Universal Robots PolyScope program: jerry_robot_1.urp

Program jerry_robot_1 (installation=default directory=/programs createdIn=5.11.9.1010452 lastSavedIn=5.11.9.1010452 robotSerialNumber=20225200364)
Calibrated DH parameters: a=[0.00002, -0.569483, -0.54992, -0.00001, -0.000036, 0]; d=[0.180894, -146.691669, 192.918669, -46.053088, 0.119778, 0.115602]; alpha=[1.571425, -0.001534, 0.003359, 1.568739, -1.571477, 0]; deltaTheta=[0, 0.376258, -0.101074, -0.275185, -0.000002, 0]
Robot Program (runOnlyOnce=false)
  Script file /programs/usbdisk/UR/jerry_new_robot_2.script
    | def Machining2():
    |   # Default parameters:
    |   global speed_ms = 0.3
    |   global speed_rads = 0.75
    |   global accel_mss = 3
    |   global accel_radss = 1.2
    |   global blend_radius_m = 0.0003
    | 
    |   # Add subprograms here
    |   # Start of main program
    |   # Program generated by RoboDK v5.6.8 for UR10e on 15/12/2023 16:19:10
    |   # Using nominal kinematics.
    |   blend_radius_m = 0.0003
    |   speed_ms = 0.01
    |   # set_reference(p[0.405000, -0.105000, 0.002000, 0.000000, 0.000000, 0.000000])
    |   set_tcp(p[0.000000, 0.000000, 0.252000, 0.000000, 0.000000, 0.000000])
    |   # Show Tool
    |   movej([0.340820, -1.401012, -2.442590, -0.868787, 1.570796, 1.911616],accel_radss,speed_rads,0,blend_radius_m)
    |   movel([0.340820, -1.453448, -2.472410, -0.786531, 1.570796, 1.911616],accel_mss,speed_ms,0,blend_radius_m)
    |   speed_ms = 0.01
    |   movel([0.340820, -1.476287, -2.483478, -0.752624, 1.570796, 1.911616],accel_mss,speed_ms,0,blend_radius_m)
    |   speed_ms = 0.003
    |   movel([0.340820, -1.485129, -2.487495, -0.739765, 1.570796, 1.911616],accel_mss,speed_ms,0,blend_radius_m)
    |   speed_ms = 0.007
    |   movel([0.329121, -1.487754, -2.485222, -0.739413, 1.570796, 1.899918],accel_mss,speed_ms,0,blend_radius_m)
    |   movel([0.326624, -1.484406, -2.488119, -0.739864, 1.570796, 1.897421],accel_mss,speed_ms,0,blend_radius_m)
    |   movel([0.324102, -1.481056, -2.491001, -0.740332, 1.570796, 1.894899],accel_mss,speed_ms,0,blend_radius_m)
    |   movel([0.325153, -1.479428, -2.492395, -0.740566, 1.570796, 1.895949],accel_mss,speed_ms,0,blend_radius_m)
    |   movel([0.326209, -1.477797, -2.493787, -0.740805, 1.570796, 1.897005],accel_mss,speed_ms,0,blend_radius_m)
    |   movel([0.325032, -1.477528, -2.494017, -0.740845, 1.570796, 1.895828],accel_mss,speed_ms,0,blend_radius_m)
    |   movel([0.324303, -1.477370, -2.494151, -0.740868, 1.570796, 1.895099],accel_mss,speed_ms,0,blend_radius_m)
    |   movel([0.315110, -1.475621, -2.495639, -0.741130, 1.570796, 1.885906],accel_mss,speed_ms,0,blend_radius_m)
    |   movel([0.311619, -1.474970, -2.496191, -0.741228, 1.570796, 1.882415],accel_mss,speed_ms,0,blend_radius_m)
    |   movel([0.310032, -1.474668, -2.496447, -0.741274, 1.570796, 1.880828],accel_mss,speed_ms,0,blend_radius_m)
    |   movel([0.308452, -1.474355, -2.496712, -0.741322, 1.570796, 1.879249],accel_mss,speed_ms,0,blend_radius_m)
    |   movel([0.306876, -1.474033, -2.496985, -0.741371, 1.570796, 1.877673],accel_mss,speed_ms,0,blend_radius_m)
    |   movel([0.305660, -1.473769, -2.497208, -0.741412, 1.570796, 1.876456],accel_mss,speed_ms,0,blend_radius_m)
    |   movel([0.304453, -1.473494, -2.497441, -0.741454, 1.570796, 1.875249],accel_mss,speed_ms,0,blend_radius_m)
    |   movel([0.303253, -1.473205, -2.497685, -0.741499, 1.570796, 1.874050],accel_mss,speed_ms,0,blend_radius_m)
    |   movel([0.302430, -1.472998, -2.497860, -0.741531, 1.570796, 1.873226],accel_mss,speed_ms,0,blend_radius_m)
    |   movel([0.301614, -1.472780, -2.498045, -0.741565, 1.570796, 1.872410],accel_mss,speed_ms,0,blend_radius_m)
    |   movel([0.300804, -1.472554, -2.498235, -0.741600, 1.570796, 1.871600],accel_mss,speed_ms,0,blend_radius_m)
    |   movel([0.299999, -1.472319, -2.498434, -0.741636, 1.570796, 1.870795],accel_mss,speed_ms,0,blend_radius_m)
    |   movel([0.299265, -1.472091, -2.498626, -0.741672, 1.570796, 1.870061],accel_mss,speed_ms,0,blend_radius_m)
    |   movel([0.298537, -1.471853, -2.498826, -0.741709, 1.570796, 1.869333],accel_mss,speed_ms,0,blend_radius_m)
    |   movel([0.297819, -1.471604, -2.499036, -0.741748, 1.570796, 1.868615],accel_mss,speed_ms,0,blend_radius_m)
    |   movel([0.297109, -1.471344, -2.499256, -0.741789, 1.570796, 1.867905],accel_mss,speed_ms,0,blend_radius_m)
    |   movel([0.296406, -1.471071, -2.499485, -0.741832, 1.570796, 1.867203],accel_mss,speed_ms,0,blend_radius_m)
    |   movel([0.295713, -1.470789, -2.499723, -0.741877, 1.570796, 1.866509],accel_mss,speed_ms,0,blend_radius_m)
    |   movel([0.295027, -1.470496, -2.499970, -0.741924, 1.570796, 1.865823],accel_mss,speed_ms,0,blend_radius_m)
    |   movel([0.294528, -1.470268, -2.500162, -0.741960, 1.570796, 1.865325],accel_mss,speed_ms,0,blend_radius_m)
    |   movel([0.294040, -1.470028, -2.500363, -0.741998, 1.570796, 1.864837],accel_mss,speed_ms,0,blend_radius_m)
    |   movel([0.293562, -1.469778, -2.500573, -0.742038, 1.570796, 1.864358],accel_mss,speed_ms,0,blend_radius_m)
    |   movel([0.293093, -1.469515, -2.500794, -0.742080, 1.570796, 1.863889],accel_mss,speed_ms,0,blend_radius_m)
    |   movel([0.292636, -1.469241, -2.501024, -0.742124, 1.570796, 1.863432],accel_mss,speed_ms,0,blend_radius_m)
    |   movel([0.292189, -1.468954, -2.501264, -0.742170, 1.570796, 1.862986],accel_mss,speed_ms,0,blend_radius_m)
    |   movel([0.291754, -1.468657, -2.501513, -0.742218, 1.570796, 1.862551],accel_mss,speed_ms,0,blend_radius_m)
    |   movel([0.291328, -1.468350, -2.501771, -0.742268, 1.570796, 1.862125],accel_mss,speed_ms,0,blend_radius_m)
    |   movel([0.290973, -1.468072, -2.502004, -0.742313, 1.570796, 1.861769],accel_mss,speed_ms,0,blend_radius_m)
    |   movel([0.290628, -1.467784, -2.502245, -0.742360, 1.570796, 1.861425],accel_mss,speed_ms,0,blend_radius_m)
    |   movel([0.290296, -1.467485, -2.502495, -0.742409, 1.570796, 1.861092],accel_mss,speed_ms,0,blend_radius_m)
    |   movel([0.289978, -1.467174, -2.502755, -0.742460, 1.570796, 1.860774],accel_mss,speed_ms,0,blend_radius_m)
    |   movel([0.289671, -1.466852, -2.503024, -0.742513, 1.570796, 1.860467],accel_mss,speed_ms,0,blend_radius_m)
    |   movel([0.289378, -1.466522, -2.503300, -0.742567, 1.570796, 1.860174],accel_mss,speed_ms,0,blend_radius_m)
    |   movel([0.289096, -1.466178, -2.503587, -0.742624, 1.570796, 1.859893],accel_mss,speed_ms,0,blend_radius_m)
    |   movel([0.288831, -1.465826, -2.503881, -0.742682, 1.570796, 1.859627],accel_mss,speed_ms,0,blend_radius_m)
    |   movel([0.288626, -1.465531, -2.504127, -0.742731, 1.570796, 1.859423],accel_mss,speed_ms,0,blend_radius_m)
    |   movel([0.288435, -1.465229, -2.504378, -0.742782, 1.570796, 1.859231],accel_mss,speed_ms,0,blend_radius_m)
    |   movel([0.288257, -1.464916, -2.504639, -0.742834, 1.570796, 1.859053],accel_mss,speed_ms,0,blend_radius_m)
    |   movel([0.288092, -1.464594, -2.504907, -0.742888, 1.570796, 1.858889],accel_mss,speed_ms,0,blend_radius_m)
    |   movel([0.287941, -1.464265, -2.505180, -0.742944, 1.570796, 1.858737],accel_mss,speed_ms,0,blend_radius_m)
    |   movel([0.287804, -1.463927, -2.505461, -0.743001, 1.570796, 1.858601],accel_mss,speed_ms,0,blend_radius_m)
    |   movel([0.287681, -1.463581, -2.505749, -0.743059, 1.570796, 1.858478],accel_mss,speed_ms,0,blend_radius_m)
    |   movel([0.287573, -1.463229, -2.506041, -0.743119, 1.570796, 1.858369],accel_mss,speed_ms,0,blend_radius_m)
    |   movel([0.287477, -1.462868, -2.506341, -0.743181, 1.570796, 1.858274],accel_mss,speed_ms,0,blend_radius_m)
    |   movel([0.287403, -1.462513, -2.506635, -0.743241, 1.570796, 1.858200],accel_mss,speed_ms,0,blend_radius_m)
    |   movel([0.287345, -1.462148, -2.506937, -0.743304, 1.570796, 1.858141],accel_mss,speed_ms,0,blend_radius_m)
    |   movel([0.287305, -1.461779, -2.507243, -0.743367, 1.570796, 1.858101],accel_mss,speed_ms,0,blend_radius_m)
    |   movel([0.287282, -1.461401, -2.507555, -0.743433, 1.570796, 1.858079],accel_mss,speed_ms,0,blend_radius_m)
    |   movel([0.287278, -1.461018, -2.507872, -0.743499, 1.570796, 1.858075],accel_mss,speed_ms,0,blend_radius_m)
    |   movel([0.287291, -1.460591, -2.508225, -0.743573, 1.570796, 1.858087],accel_mss,speed_ms,0,blend_radius_m)
    |   movel([0.287320, -1.460158, -2.508582, -0.743649, 1.570796, 1.858116],accel_mss,speed_ms,0,blend_radius_m)
    |   movel([0.287362, -1.459724, -2.508940, -0.743725, 1.570796, 1.858158],accel_mss,speed_ms,0,blend_radius_m)
    |   movel([0.287419, -1.459283, -2.509304, -0.743802, 1.570796, 1.858216],accel_mss,speed_ms,0,blend_radius_m)
    |   movel([0.287492, -1.458840, -2.509669, -0.743881, 1.570796, 1.858288],accel_mss,speed_ms,0,blend_radius_m)
    |   movel([0.287580, -1.458381, -2.510046, -0.743962, 1.570796, 1.858377],accel_mss,speed_ms,0,blend_radius_m)
    |   movel([0.287685, -1.457918, -2.510427, -0.744044, 1.570796, 1.858482],accel_mss,speed_ms,0,blend_radius_m)
    |   movel([0.287806, -1.457452, -2.510809, -0.744128, 1.570796, 1.858602],accel_mss,speed_ms,0,blend_radius_m)
    |   movel([0.287939, -1.456985, -2.511192, -0.744211, 1.570796, 1.858736],accel_mss,speed_ms,0,blend_radius_m)
    |   movel([0.288089, -1.456515, -2.511578, -0.744296, 1.570796, 1.858886],accel_mss,speed_ms,0,blend_radius_m)
    |   movel([0.288247, -1.456059, -2.511951, -0.744379, 1.570796, 1.859044],accel_mss,speed_ms,0,blend_radius_m)
    |   movel([0.288421, -1.455602, -2.512326, -0.744462, 1.570796, 1.859217],accel_mss,speed_ms,0,blend_radius_m)
    |   movel([0.288612, -1.455142, -2.512701, -0.744545, 1.570796, 1.859408],accel_mss,speed_ms,0,blend_radius_m)
    |   movel([0.288815, -1.454686, -2.513074, -0.744629, 1.570796, 1.859612],accel_mss,speed_ms,0,blend_radius_m)
    |   movel([0.289034, -1.454228, -2.513449, -0.744713, 1.570796, 1.859831],accel_mss,speed_ms,0,blend_radius_m)
    |   movel([0.289272, -1.453758, -2.513832, -0.744800, 1.570796, 1.860068],accel_mss,speed_ms,0,blend_radius_m)
    |   movel([0.289521, -1.453288, -2.514214, -0.744886, 1.570796, 1.860317],accel_mss,speed_ms,0,blend_radius_m)
    |   movel([0.289777, -1.452822, -2.514594, -0.744973, 1.570796, 1.860573],accel_mss,speed_ms,0,blend_radius_m)
    |   movel([0.290044, -1.452355, -2.514974, -0.745060, 1.570796, 1.860841],accel_mss,speed_ms,0,blend_radius_m)
    |   movel([0.290115, -1.452249, -2.515060, -0.745080, 1.570796, 1.860912],accel_mss,speed_ms,0,blend_radius_m)
    |   movel([0.290197, -1.452143, -2.515146, -0.745100, 1.570796, 1.860993],accel_mss,speed_ms,0,blend_radius_m)
    |   movel([0.290291, -1.452045, -2.515226, -0.745118, 1.570796, 1.861087],accel_mss,speed_ms,0,blend_radius_m)
    |   movel([0.290394, -1.451953, -2.515300, -0.745135, 1.570796, 1.861190],accel_mss,speed_ms,0,blend_radius_m)
    |   movel([0.290502, -1.451871, -2.515367, -0.745151, 1.570796, 1.861298],accel_mss,speed_ms,0,blend_radius_m)
    |   movel([0.290618, -1.451797, -2.515428, -0.745165, 1.570796, 1.861415],accel_mss,speed_ms,0,blend_radius_m)
    |   movel([0.290740, -1.451733, -2.515479, -0.745177, 1.570796, 1.861536],accel_mss,speed_ms,0,blend_radius_m)
    |   movel([0.290896, -1.451667, -2.515533, -0.745189, 1.570796, 1.861693],accel_mss,speed_ms,0,blend_radius_m)
    |   movel([0.291052, -1.451616, -2.515574, -0.745199, 1.570796, 1.861849],accel_mss,speed_ms,0,blend_radius_m)
    |   movel([0.291206, -1.451580, -2.515603, -0.745205, 1.570796, 1.862002],accel_mss,speed_ms,0,blend_radius_m)
    |   movel([0.291358, -1.451560, -2.515620, -0.745209, 1.570796, 1.862155],accel_mss,speed_ms,0,blend_radius_m)
    |   movel([0.291506, -1.451555, -2.515624, -0.745210, 1.570796, 1.862302],accel_mss,speed_ms,0,blend_radius_m)
    |   movel([0.291645, -1.451567, -2.515614, -0.745208, 1.570796, 1.862442],accel_mss,speed_ms,0,blend_radius_m)
    |   movel([0.292393, -1.451683, -2.515520, -0.745186, 1.570796, 1.863189],accel_mss,speed_ms,0,blend_radius_m)
    |   movel([0.293133, -1.451812, -2.515415, -0.745162, 1.570796, 1.863929],accel_mss,speed_ms,0,blend_radius_m)
    |   movel([0.293865, -1.451954, -2.515299, -0.745135, 1.570796, 1.864661],accel_mss,speed_ms,0,blend_radius_m)
    |   movel([0.294949, -1.452176, -2.515120, -0.745094, 1.570796, 1.865746],accel_mss,speed_ms,0,blend_radius_m)
    |   movel([0.295293, -1.451133, -2.515966, -0.745290, 1.570796, 1.866090],accel_mss,speed_ms,0,blend_radius_m)
    |   movel([0.295639, -1.450087, -2.516814, -0.745488, 1.570796, 1.866435],accel_mss,speed_ms,0,blend_radius_m)
    |   movel([0.271091, -1.452301, -2.515018, -0.745070, 1.570796, 1.841887],accel_mss,speed_ms,0,blend_radius_m)
    |   movel([0.256701, -1.453830, -2.513773, -0.744786, 1.570796, 1.827497],accel_mss,speed_ms,0,blend_radius_m)
    |   movel([0.253581, -1.454176, -2.513491, -0.744722, 1.570796, 1.824377],accel_mss,speed_ms,0,blend_radius_m)
    |   movel([0.250464, -1.454516, -2.513213, -0.744660, 1.570796, 1.821261],accel_mss,speed_ms,0,blend_radius_m)
    |   movel([0.248542, -1.454722, -2.513045, -0.744622, 1.570796, 1.819338],accel_mss,speed_ms,0,blend_radius_m)
    |   movel([0.246618, -1.454926, -2.512878, -0.744585, 1.570796, 1.817414],accel_mss,speed_ms,0,blend_radius_m)
    |   movel([0.246504, -1.454932, -2.512873, -0.744584, 1.570796, 1.817301],accel_mss,speed_ms,0,blend_radius_m)
    |   movel([0.246399, -1.454926, -2.512878, -0.744585, 1.570796, 1.817195],accel_mss,speed_ms,0,blend_radius_m)
    |   movel([0.246297, -1.454907, -2.512894, -0.744588, 1.570796, 1.817093],accel_mss,speed_ms,0,blend_radius_m)
    |   movel([0.246204, -1.454876, -2.512919, -0.744594, 1.570796, 1.817001],accel_mss,speed_ms,0,blend_radius_m)
    |   movel([0.246122, -1.454833, -2.512954, -0.744602, 1.570796, 1.816918],accel_mss,speed_ms,0,blend_radius_m)
    |   movel([0.246053, -1.454780, -2.512998, -0.744612, 1.570796, 1.816849],accel_mss,speed_ms,0,blend_radius_m)
    |   movel([0.246000, -1.454714, -2.513051, -0.744624, 1.570796, 1.816796],accel_mss,speed_ms,0,blend_radius_m)
    |   movel([0.245961, -1.454638, -2.513114, -0.744638, 1.570796, 1.816758],accel_mss,speed_ms,0,blend_radius_m)
    |   movel([0.245935, -1.454548, -2.513187, -0.744654, 1.570796, 1.816731],accel_mss,speed_ms,0,blend_radius_m)
    |   movel([0.245925, -1.454450, -2.513267, -0.744672, 1.570796, 1.816722],accel_mss,speed_ms,0,blend_radius_m)
    |   movel([0.245930, -1.454348, -2.513350, -0.744691, 1.570796, 1.816726],accel_mss,speed_ms,0,blend_radius_m)
    |   movel([0.245955, -1.454173, -2.513493, -0.744723, 1.570796, 1.816751],accel_mss,speed_ms,0,blend_radius_m)
    |   movel([0.245990, -1.453994, -2.513639, -0.744756, 1.570796, 1.816786],accel_mss,speed_ms,0,blend_radius_m)
    |   movel([0.246033, -1.453813, -2.513786, -0.744789, 1.570796, 1.816830],accel_mss,speed_ms,0,blend_radius_m)
    |   movel([0.246212, -1.453141, -2.514334, -0.744914, 1.570796, 1.817008],accel_mss,speed_ms,0,blend_radius_m)
    |   movel([0.246397, -1.452468, -2.514882, -0.745039, 1.570796, 1.817193],accel_mss,speed_ms,0,blend_radius_m)
    |   movel([0.247002, -1.450297, -2.516644, -0.745448, 1.570796, 1.817798],accel_mss,speed_ms,0,blend_radius_m)
    |   movel([0.232327, -1.452185, -2.515112, -0.745092, 1.570796, 1.803123],accel_mss,speed_ms,0,blend_radius_m)
    |   movel([0.217636, -1.454249, -2.513431, -0.744709, 1.570796, 1.788433],accel_mss,speed_ms,0,blend_radius_m)
    |   movel([0.217419, -1.455129, -2.512713, -0.744548, 1.570796, 1.788215],accel_mss,speed_ms,0,blend_radius_m)
    |   movel([0.217201, -1.456007, -2.511994, -0.744388, 1.570796, 1.787998],accel_mss,speed_ms,0,blend_radius_m)
    |   movel([0.191731, -1.459985, -2.508725, -0.743679, 1.570796, 1.762527],accel_mss,speed_ms,0,blend_radius_m)
    |   movel([0.166263, -1.464470, -2.505010, -0.742909, 1.570796, 1.737059],accel_mss,speed_ms,0,blend_radius_m)
    |   movel([0.164813, -1.465408, -2.504229, -0.742752, 1.570796, 1.735609],accel_mss,speed_ms,0,blend_radius_m)
    |   movel([0.164370, -1.465688, -2.503995, -0.742705, 1.570796, 1.735166],accel_mss,speed_ms,0,blend_radius_m)
    |   movel([0.163922, -1.465960, -2.503769, -0.742660, 1.570796, 1.734718],accel_mss,speed_ms,0,blend_radius_m)
    |   movel([0.163472, -1.466223, -2.503549, -0.742617, 1.570796, 1.734268],accel_mss,speed_ms,0,blend_radius_m)
    |   movel([0.162985, -1.466498, -2.503320, -0.742571, 1.570796, 1.733782],accel_mss,speed_ms,0,blend_radius_m)
    |   movel([0.162497, -1.466763, -2.503099, -0.742527, 1.570796, 1.733293],accel_mss,speed_ms,0,blend_radius_m)
    |   movel([0.162003, -1.467023, -2.502881, -0.742485, 1.570796, 1.732799],accel_mss,speed_ms,0,blend_radius_m)
    |   movel([0.161497, -1.467278, -2.502668, -0.742443, 1.570796, 1.732293],accel_mss,speed_ms,0,blend_radius_m)
    |   movel([0.160989, -1.467526, -2.502461, -0.742402, 1.570796, 1.731785],accel_mss,speed_ms,0,blend_radius_m)
    |   movel([0.160477, -1.467767, -2.502259, -0.742363, 1.570796, 1.731274],accel_mss,speed_ms,0,blend_radius_m)
    |   movel([0.159975, -1.467993, -2.502070, -0.742326, 1.570796, 1.730772],accel_mss,speed_ms,0,blend_radius_m)
    |   movel([0.159473, -1.468210, -2.501888, -0.742291, 1.570796, 1.730269],accel_mss,speed_ms,0,blend_radius_m)
    |   movel([0.158968, -1.468419, -2.501714, -0.742257, 1.570796, 1.729765],accel_mss,speed_ms,0,blend_radius_m)
    |   movel([0.158596, -1.468562, -2.501593, -0.742234, 1.570796, 1.729392],accel_mss,speed_ms,0,blend_radius_m)
    |   movel([0.158224, -1.468695, -2.501482, -0.742212, 1.570796, 1.729020],accel_mss,speed_ms,0,blend_radius_m)
    |   movel([0.157852, -1.468815, -2.501381, -0.742193, 1.570796, 1.728648],accel_mss,speed_ms,0,blend_radius_m)
    |   movel([0.157477, -1.468924, -2.501290, -0.742175, 1.570796, 1.728274],accel_mss,speed_ms,0,blend_radius_m)
    |   movel([0.156691, -1.469135, -2.501113, -0.742141, 1.570796, 1.727488],accel_mss,speed_ms,0,blend_radius_m)
    |   movel([0.155905, -1.469336, -2.500944, -0.742109, 1.570796, 1.726702],accel_mss,speed_ms,0,blend_radius_m)
    |   movel([0.155121, -1.469529, -2.500782, -0.742078, 1.570796, 1.725917],accel_mss,speed_ms,0,blend_radius_m)
    |   movel([0.153917, -1.469812, -2.500544, -0.742032, 1.570796, 1.724713],accel_mss,speed_ms,0,blend_radius_m)
    |   movel([0.152713, -1.470086, -2.500314, -0.741989, 1.570796, 1.723509],accel_mss,speed_ms,0,blend_radius_m)
    |   movel([0.152591, -1.470106, -2.500298, -0.741986, 1.570796, 1.723388],accel_mss,speed_ms,0,blend_radius_m)
    |   movel([0.152472, -1.470112, -2.500292, -0.741985, 1.570796, 1.723268],accel_mss,speed_ms,0,blend_radius_m)
    |   movel([0.152357, -1.470105, -2.500299, -0.741986, 1.570796, 1.723154],accel_mss,speed_ms,0,blend_radius_m)
    |   movel([0.152251, -1.470084, -2.500316, -0.741989, 1.570796, 1.723048],accel_mss,speed_ms,0,blend_radius_m)
    |   movel([0.152157, -1.470049, -2.500346, -0.741995, 1.570796, 1.722953],accel_mss,speed_ms,0,blend_radius_m)
    |   movel([0.152111, -1.470019, -2.500371, -0.741999, 1.570796, 1.722907],accel_mss,speed_ms,0,blend_radius_m)
    |   movel([0.152079, -1.469978, -2.500405, -0.742006, 1.570796, 1.722875],accel_mss,speed_ms,0,blend_radius_m)
    |   movel([0.152064, -1.469927, -2.500448, -0.742014, 1.570796, 1.722861],accel_mss,speed_ms,0,blend_radius_m)
    |   movel([0.152066, -1.469869, -2.500497, -0.742023, 1.570796, 1.722862],accel_mss,speed_ms,0,blend_radius_m)
    |   movel([0.152646, -1.466186, -2.503580, -0.742623, 1.570796, 1.723442],accel_mss,speed_ms,0,blend_radius_m)
    |   movel([0.153067, -1.463577, -2.505752, -0.743060, 1.570796, 1.723863],accel_mss,speed_ms,0,blend_radius_m)
    |   movel([0.153505, -1.460953, -2.507926, -0.743510, 1.570796, 1.724301],accel_mss,speed_ms,0,blend_radius_m)
    |   movel([0.154303, -1.456267, -2.511781, -0.744341, 1.570796, 1.725099],accel_mss,speed_ms,0,blend_radius_m)
    |   movel([0.155114, -1.451549, -2.515629, -0.745211, 1.570796, 1.725910],accel_mss,speed_ms,0,blend_radius_m)
    |   movel([0.158413, -1.432638, -2.530710, -0.749041, 1.570796, 1.729209],accel_mss,speed_ms,0,blend_radius_m)
    |   movel([0.159001, -1.432517, -2.530805, -0.749067, 1.570796, 1.729798],accel_mss,speed_ms,0,blend_radius_m)
    |   movel([0.159337, -1.432432, -2.530871, -0.749086, 1.570796, 1.730133],accel_mss,speed_ms,0,blend_radius_m)
    |   movel([0.159426, -1.432396, -2.530899, -0.749094, 1.570796, 1.730223],accel_mss,speed_ms,0,blend_radius_m)
    |   movel([0.159506, -1.432338, -2.530944, -0.749106, 1.570796, 1.730303],accel_mss,speed_ms,0,blend_radius_m)
    |   movel([0.159568, -1.432271, -2.530997, -0.749121, 1.570796, 1.730364],accel_mss,speed_ms,0,blend_radius_m)
    |   movel([0.159606, -1.432196, -2.531056, -0.749137, 1.570796, 1.730403],accel_mss,speed_ms,0,blend_radius_m)
    |   movel([0.159676, -1.431929, -2.531265, -0.749195, 1.570796, 1.730472],accel_mss,speed_ms,0,blend_radius_m)
    |   movel([0.159710, -1.431790, -2.531374, -0.749226, 1.570796, 1.730506],accel_mss,speed_ms,0,blend_radius_m)
    |   movel([0.159761, -1.431646, -2.531486, -0.749257, 1.570796, 1.730557],accel_mss,speed_ms,0,blend_radius_m)
    |   movel([0.159794, -1.431588, -2.531532, -0.749270, 1.570796, 1.730591],accel_mss,speed_ms,0,blend_radius_m)
    |   movel([0.159840, -1.431533, -2.531574, -0.749282, 1.570796, 1.730636],accel_mss,speed_ms,0,blend_radius_m)
    |   movel([0.159898, -1.431484, -2.531613, -0.749292, 1.570796, 1.730695],accel_mss,speed_ms,0,blend_radius_m)
    |   movel([0.159982, -1.431433, -2.531652, -0.749303, 1.570796, 1.730778],accel_mss,speed_ms,0,blend_radius_m)
    |   movel([0.160068, -1.431390, -2.531686, -0.749313, 1.570796, 1.730864],accel_mss,speed_ms,0,blend_radius_m)
    |   movel([0.160157, -1.431358, -2.531711, -0.749320, 1.570796, 1.730953],accel_mss,speed_ms,0,blend_radius_m)
    |   movel([0.160485, -1.431253, -2.531793, -0.749343, 1.570796, 1.731282],accel_mss,speed_ms,0,blend_radius_m)
    |   movel([0.160815, -1.431156, -2.531869, -0.749364, 1.570796, 1.731611],accel_mss,speed_ms,0,blend_radius_m)
    |   movel([0.161117, -1.431073, -2.531934, -0.749382, 1.570796, 1.731914],accel_mss,speed_ms,0,blend_radius_m)
    |   movel([0.161418, -1.431000, -2.531991, -0.749398, 1.570796, 1.732214],accel_mss,speed_ms,0,blend_radius_m)
    |   movel([0.161719, -1.430934, -2.532042, -0.749413, 1.570796, 1.732515],accel_mss,speed_ms,0,blend_radius_m)
    |   movel([0.162016, -1.430880, -2.532085, -0.749425, 1.570796, 1.732812],accel_mss,speed_ms,0,blend_radius_m)
    |   movel([0.162543, -1.430796, -2.532150, -0.749443, 1.570796, 1.733339],accel_mss,speed_ms,0,blend_radius_m)
    |   movel([0.163067, -1.430723, -2.532207, -0.749459, 1.570796, 1.733864],accel_mss,speed_ms,0,blend_radius_m)
    |   movel([0.163588, -1.430661, -2.532256, -0.749473, 1.570796, 1.734384],accel_mss,speed_ms,0,blend_radius_m)
    |   movel([0.164138, -1.430604, -2.532299, -0.749485, 1.570796, 1.734935],accel_mss,speed_ms,0,blend_radius_m)
    |   movel([0.164685, -1.430557, -2.532336, -0.749496, 1.570796, 1.735481],accel_mss,speed_ms,0,blend_radius_m)
    |   movel([0.165227, -1.430523, -2.532363, -0.749503, 1.570796, 1.736023],accel_mss,speed_ms,0,blend_radius_m)
    |   movel([0.165710, -1.430504, -2.532377, -0.749507, 1.570796, 1.736506],accel_mss,speed_ms,0,blend_radius_m)
    |   movel([0.166191, -1.430497, -2.532384, -0.749509, 1.570796, 1.736987],accel_mss,speed_ms,0,blend_radius_m)
    |   movel([0.166662, -1.430503, -2.532379, -0.749508, 1.570796, 1.737459],accel_mss,speed_ms,0,blend_radius_m)
    |   movel([0.167080, -1.430522, -2.532364, -0.749503, 1.570796, 1.737876],accel_mss,speed_ms,0,blend_radius_m)
    |   movel([0.167490, -1.430556, -2.532337, -0.749496, 1.570796, 1.738286],accel_mss,speed_ms,0,blend_radius_m)
    |   movel([0.167893, -1.430602, -2.532301, -0.749486, 1.570796, 1.738689],accel_mss,speed_ms,0,blend_radius_m)
    |   movel([0.168370, -1.430673, -2.532246, -0.749470, 1.570796, 1.739166],accel_mss,speed_ms,0,blend_radius_m)
    |   movel([0.168842, -1.430753, -2.532184, -0.749453, 1.570796, 1.739639],accel_mss,speed_ms,0,blend_radius_m)
    |   movel([0.169308, -1.430842, -2.532114, -0.749433, 1.570796, 1.740105],accel_mss,speed_ms,0,blend_radius_m)
    |   movel([0.169772, -1.430941, -2.532036, -0.749411, 1.570796, 1.740569],accel_mss,speed_ms,0,blend_radius_m)
    |   movel([0.170227, -1.431051, -2.531951, -0.749387, 1.570796, 1.741024],accel_mss,speed_ms,0,blend_radius_m)
    |   movel([0.170676, -1.431169, -2.531858, -0.749361, 1.570796, 1.741472],accel_mss,speed_ms,0,blend_radius_m)
    |   movel([0.171046, -1.431280, -2.531772, -0.749337, 1.570796, 1.741842],accel_mss,speed_ms,0,blend_radius_m)
    |   movel([0.171404, -1.431403, -2.531676, -0.749310, 1.570796, 1.742200],accel_mss,speed_ms,0,blend_radius_m)
    |   movel([0.171754, -1.431541, -2.531568, -0.749280, 1.570796, 1.742551],accel_mss,speed_ms,0,blend_radius_m)
    |   movel([0.172514, -1.431858, -2.531320, -0.749211, 1.570796, 1.743310],accel_mss,speed_ms,0,blend_radius_m)
    |   movel([0.199133, -1.426954, -2.535137, -0.750298, 1.570796, 1.769929],accel_mss,speed_ms,0,blend_radius_m)
    |   movel([0.225758, -1.422602, -2.538494, -0.751293, 1.570796, 1.796555],accel_mss,speed_ms,0,blend_radius_m)
    |   movel([0.225503, -1.423608, -2.537721, -0.751061, 1.570796, 1.796299],accel_mss,speed_ms,0,blend_radius_m)
    |   movel([0.225247, -1.424612, -2.536947, -0.750830, 1.570796, 1.796044],accel_mss,speed_ms,0,blend_radius_m)
    |   movel([0.232573, -1.423517, -2.537791, -0.751082, 1.570796, 1.803369],accel_mss,speed_ms,0,blend_radius_m)
    |   movel([0.237752, -1.422744, -2.538385, -0.751260, 1.570796, 1.808548],accel_mss,speed_ms,0,blend_radius_m)
    |   movel([0.239900, -1.422404, -2.538646, -0.751339, 1.570796, 1.810696],accel_mss,speed_ms,0,blend_radius_m)
    |   movel([0.239919, -1.422377, -2.538667, -0.751345, 1.570796, 1.810715],accel_mss,speed_ms,0,blend_radius_m)
    |   movel([0.239924, -1.422315, -2.538714, -0.751360, 1.570796, 1.810720],accel_mss,speed_ms,0,blend_radius_m)
    |   movel([0.239692, -1.420997, -2.539724, -0.751667, 1.570796, 1.810489],accel_mss,speed_ms,0,blend_radius_m)
    |   movel([0.239636, -1.420602, -2.540027, -0.751760, 1.570796, 1.810432],accel_mss,speed_ms,0,blend_radius_m)
    |   movel([0.239597, -1.420198, -2.540336, -0.751855, 1.570796, 1.810393],accel_mss,speed_ms,0,blend_radius_m)
    |   movel([0.239576, -1.419811, -2.540632, -0.751946, 1.570796, 1.810372],accel_mss,speed_ms,0,blend_radius_m)
    |   movel([0.239572, -1.419418, -2.540932, -0.752039, 1.570796, 1.810368],accel_mss,speed_ms,0,blend_radius_m)
    |   movel([0.239586, -1.419018, -2.541237, -0.752134, 1.570796, 1.810382],accel_mss,speed_ms,0,blend_radius_m)
    |   movel([0.239616, -1.418605, -2.541552, -0.752232, 1.570796, 1.810413],accel_mss,speed_ms,0,blend_radius_m)
    |   movel([0.239666, -1.418187, -2.541870, -0.752332, 1.570796, 1.810462],accel_mss,speed_ms,0,blend_radius_m)
    |   movel([0.239730, -1.417764, -2.542192, -0.752433, 1.570796, 1.810527],accel_mss,speed_ms,0,blend_radius_m)
    |   movel([0.239821, -1.417295, -2.542549, -0.752545, 1.570796, 1.810617],accel_mss,speed_ms,0,blend_radius_m)
    |   movel([0.239923, -1.416824, -2.542907, -0.752658, 1.570796, 1.810719],accel_mss,speed_ms,0,blend_radius_m)
    |   movel([0.240041, -1.416350, -2.543266, -0.752772, 1.570796, 1.810838],accel_mss,speed_ms,0,blend_radius_m)
    |   movel([0.240151, -1.415951, -2.543569, -0.752869, 1.570796, 1.810947],accel_mss,speed_ms,0,blend_radius_m)
    |   movel([0.240276, -1.415547, -2.543875, -0.752967, 1.570796, 1.811072],accel_mss,speed_ms,0,blend_radius_m)
    |   movel([0.240409, -1.415144, -2.544180, -0.753064, 1.570796, 1.811205],accel_mss,speed_ms,0,blend_radius_m)
    |   movel([0.240556, -1.414739, -2.544487, -0.753163, 1.570796, 1.811353],accel_mss,speed_ms,0,blend_radius_m)
    |   movel([0.240701, -1.414371, -2.544766, -0.753253, 1.570796, 1.811497],accel_mss,speed_ms,0,blend_radius_m)
    |   movel([0.240859, -1.414002, -2.545044, -0.753343, 1.570796, 1.811655],accel_mss,speed_ms,0,blend_radius_m)
    |   movel([0.241032, -1.413633, -2.545322, -0.753433, 1.570796, 1.811829],accel_mss,speed_ms,0,blend_radius_m)
    |   movel([0.241218, -1.413264, -2.545601, -0.753524, 1.570796, 1.812014],accel_mss,speed_ms,0,blend_radius_m)
    |   movel([0.241424, -1.412884, -2.545887, -0.753618, 1.570796, 1.812220],accel_mss,speed_ms,0,blend_radius_m)
    |   movel([0.241644, -1.412504, -2.546174, -0.753711, 1.570796, 1.812440],accel_mss,speed_ms,0,blend_radius_m)
    |   movel([0.241875, -1.412126, -2.546458, -0.753805, 1.570796, 1.812671],accel_mss,speed_ms,0,blend_radius_m)
    |   movel([0.242118, -1.411750, -2.546741, -0.753898, 1.570796, 1.812915],accel_mss,speed_ms,0,blend_radius_m)
    |   movel([0.242518, -1.411167, -2.547179, -0.754043, 1.570796, 1.813314],accel_mss,speed_ms,0,blend_radius_m)
    |   movel([0.242932, -1.410590, -2.547612, -0.754187, 1.570796, 1.813728],accel_mss,speed_ms,0,blend_radius_m)
    |   movel([0.243362, -1.410013, -2.548044, -0.754331, 1.570796, 1.814158],accel_mss,speed_ms,0,blend_radius_m)
    |   movel([0.244602, -1.408393, -2.549257, -0.754739, 1.570796, 1.815398],accel_mss,speed_ms,0,blend_radius_m)
    |   movel([0.242538, -1.408689, -2.549035, -0.754664, 1.570796, 1.813334],accel_mss,speed_ms,0,blend_radius_m)
    |   movel([0.240471, -1.408990, -2.548811, -0.754588, 1.570796, 1.811267],accel_mss,speed_ms,0,blend_radius_m)
    |   movel([0.240725, -1.408045, -2.549517, -0.754827, 1.570796, 1.811521],accel_mss,speed_ms,0,blend_radius_m)
    |   movel([0.240980, -1.407099, -2.550222, -0.755068, 1.570796, 1.811776],accel_mss,speed_ms,0,blend_radius_m)
    |   movel([0.234750, -1.408027, -2.549530, -0.754832, 1.570796, 1.805546],accel_mss,speed_ms,0,blend_radius_m)
    |   movel([0.228517, -1.408987, -2.548813, -0.754589, 1.570796, 1.799313],accel_mss,speed_ms,0,blend_radius_m)
    |   movel([0.228254, -1.410014, -2.548044, -0.754331, 1.570796, 1.799050],accel_mss,speed_ms,0,blend_radius_m)
    |   movel([0.227991, -1.411039, -2.547275, -0.754075, 1.570796, 1.798787],accel_mss,speed_ms,0,blend_radius_m)
    |   movel([0.200872, -1.415564, -2.543863, -0.752963, 1.570796, 1.771668],accel_mss,speed_ms,0,blend_radius_m)
    |   movel([0.173761, -1.420659, -2.539983, -0.751747, 1.570796, 1.744558],accel_mss,speed_ms,0,blend_radius_m)
    |   movel([0.171928, -1.421738, -2.539157, -0.751494, 1.570796, 1.742724],accel_mss,speed_ms,0,blend_radius_m)
    |   movel([0.171423, -1.422028, -2.538935, -0.751427, 1.570796, 1.742220],accel_mss,speed_ms,0,blend_radius_m)
    |   movel([0.170917, -1.422309, -2.538719, -0.751361, 1.570796, 1.741713],accel_mss,speed_ms,0,blend_radius_m)
    |   movel([0.170408, -1.422578, -2.538512, -0.751299, 1.570796, 1.741204],accel_mss,speed_ms,0,blend_radius_m)
    |   movel([0.169896, -1.422840, -2.538311, -0.751238, 1.570796, 1.740692],accel_mss,speed_ms,0,blend_radius_m)
    |   movel([0.169382, -1.423091, -2.538118, -0.751180, 1.570796, 1.740179],accel_mss,speed_ms,0,blend_radius_m)
    |   movel([0.168856, -1.423338, -2.537928, -0.751123, 1.570796, 1.739652],accel_mss,speed_ms,0,blend_radius_m)
    |   movel([0.168327, -1.423574, -2.537747, -0.751069, 1.570796, 1.739124],accel_mss,speed_ms,0,blend_radius_m)
    |   movel([0.167799, -1.423800, -2.537573, -0.751016, 1.570796, 1.738595],accel_mss,speed_ms,0,blend_radius_m)
    |   movel([0.167270, -1.424016, -2.537406, -0.750967, 1.570796, 1.738066],accel_mss,speed_ms,0,blend_radius_m)
    |   movel([0.166739, -1.424221, -2.537248, -0.750920, 1.570796, 1.737535],accel_mss,speed_ms,0,blend_radius_m)
    |   movel([0.166217, -1.424414, -2.537099, -0.750875, 1.570796, 1.737013],accel_mss,speed_ms,0,blend_radius_m)
    |   movel([0.165695, -1.424596, -2.536959, -0.750834, 1.570796, 1.736492],accel_mss,speed_ms,0,blend_radius_m)
    |   movel([0.165174, -1.424766, -2.536828, -0.750795, 1.570796, 1.735970],accel_mss,speed_ms,0,blend_radius_m)
    |   movel([0.164651, -1.424928, -2.536703, -0.750758, 1.570796, 1.735448],accel_mss,speed_ms,0,blend_radius_m)
    |   movel([0.164132, -1.425078, -2.536588, -0.750724, 1.570796, 1.734928],accel_mss,speed_ms,0,blend_radius_m)
    |   movel([0.163640, -1.425208, -2.536487, -0.750694, 1.570796, 1.734437],accel_mss,speed_ms,0,blend_radius_m)
    |   movel([0.163149, -1.425327, -2.536395, -0.750667, 1.570796, 1.733945],accel_mss,speed_ms,0,blend_radius_m)
    |   movel([0.162660, -1.425435, -2.536312, -0.750642, 1.570796, 1.733456],accel_mss,speed_ms,0,blend_radius_m)
    |   movel([0.162175, -1.425529, -2.536239, -0.750621, 1.570796, 1.732972],accel_mss,speed_ms,0,blend_radius_m)
    |   movel([0.161691, -1.425611, -2.536176, -0.750602, 1.570796, 1.732488],accel_mss,speed_ms,0,blend_radius_m)
    |   movel([0.161060, -1.425708, -2.536101, -0.750580, 1.570796, 1.731856],accel_mss,speed_ms,0,blend_radius_m)
    |   movel([0.160519, -1.425780, -2.536045, -0.750564, 1.570796, 1.731315],accel_mss,speed_ms,0,blend_radius_m)
    |   movel([0.160058, -1.425836, -2.536002, -0.750551, 1.570796, 1.730854],accel_mss,speed_ms,0,blend_radius_m)
    |   movel([0.160024, -1.425835, -2.536003, -0.750551, 1.570796, 1.730820],accel_mss,speed_ms,0,blend_radius_m)
    |   movel([0.160001, -1.425822, -2.536013, -0.750554, 1.570796, 1.730798],accel_mss,speed_ms,0,blend_radius_m)
    |   movel([0.159985, -1.425800, -2.536030, -0.750559, 1.570796, 1.730782],accel_mss,speed_ms,0,blend_radius_m)
    |   movel([0.159984, -1.425768, -2.536054, -0.750566, 1.570796, 1.730781],accel_mss,speed_ms,0,blend_radius_m)
    |   movel([0.160995, -1.420069, -2.540434, -0.751885, 1.570796, 1.731792],accel_mss,speed_ms,0,blend_radius_m)
    |   movel([0.162132, -1.413716, -2.545260, -0.753413, 1.570796, 1.732928],accel_mss,speed_ms,0,blend_radius_m)
    |   movel([0.163517, -1.406100, -2.550965, -0.755323, 1.570796, 1.734314],accel_mss,speed_ms,0,blend_radius_m)
    |   movel([0.167261, -1.385826, -2.565740, -0.760823, 1.570796, 1.738057],accel_mss,speed_ms,0,blend_radius_m)
    |   movel([0.167902, -1.385686, -2.565840, -0.760863, 1.570796, 1.738699],accel_mss,speed_ms,0,blend_radius_m)
    |   movel([0.168291, -1.385588, -2.565910, -0.760891, 1.570796, 1.739087],accel_mss,speed_ms,0,blend_radius_m)
    |   movel([0.168373, -1.385553, -2.565935, -0.760901, 1.570796, 1.739169],accel_mss,speed_ms,0,blend_radius_m)
    |   movel([0.168445, -1.385495, -2.565976, -0.760918, 1.570796, 1.739242],accel_mss,speed_ms,0,blend_radius_m)
    |   movel([0.168496, -1.385427, -2.566024, -0.760937, 1.570796, 1.739292],accel_mss,speed_ms,0,blend_radius_m)
    |   movel([0.168519, -1.385355, -2.566076, -0.760958, 1.570796, 1.739315],accel_mss,speed_ms,0,blend_radius_m)
    |   movel([0.168526, -1.385058, -2.566288, -0.761043, 1.570796, 1.739323],accel_mss,speed_ms,0,blend_radius_m)
    |   movel([0.168526, -1.384911, -2.566393, -0.761085, 1.570796, 1.739323],accel_mss,speed_ms,0,blend_radius_m)
    |   movel([0.168542, -1.384756, -2.566503, -0.761130, 1.570796, 1.739338],accel_mss,speed_ms,0,blend_radius_m)
    |   movel([0.168559, -1.384700, -2.566543, -0.761146, 1.570796, 1.739356],accel_mss,speed_ms,0,blend_radius_m)
    |   movel([0.168591, -1.384645, -2.566582, -0.761162, 1.570796, 1.739388],accel_mss,speed_ms,0,blend_radius_m)
    |   movel([0.168641, -1.384594, -2.566619, -0.761177, 1.570796, 1.739437],accel_mss,speed_ms,0,blend_radius_m)
    |   movel([0.168708, -1.384541, -2.566656, -0.761192, 1.570796, 1.739504],accel_mss,speed_ms,0,blend_radius_m)
    |   movel([0.168780, -1.384498, -2.566687, -0.761204, 1.570796, 1.739576],accel_mss,speed_ms,0,blend_radius_m)
    |   movel([0.168855, -1.384463, -2.566712, -0.761214, 1.570796, 1.739651],accel_mss,speed_ms,0,blend_radius_m)
    |   movel([0.169154, -1.384353, -2.566790, -0.761246, 1.570796, 1.739950],accel_mss,speed_ms,0,blend_radius_m)
    |   movel([0.169453, -1.384248, -2.566865, -0.761276, 1.570796, 1.740249],accel_mss,speed_ms,0,blend_radius_m)
    |   movel([0.169792, -1.384138, -2.566943, -0.761308, 1.570796, 1.740588],accel_mss,speed_ms,0,blend_radius_m)
    |   movel([0.170131, -1.384045, -2.567009, -0.761335, 1.570796, 1.740927],accel_mss,speed_ms,0,blend_radius_m)
    |   movel([0.170466, -1.383970, -2.567063, -0.761356, 1.570796, 1.741262],accel_mss,speed_ms,0,blend_radius_m)
    |   movel([0.170944, -1.383876, -2.567130, -0.761383, 1.570796, 1.741740],accel_mss,speed_ms,0,blend_radius_m)
    |   movel([0.171423, -1.383791, -2.567190, -0.761408, 1.570796, 1.742219],accel_mss,speed_ms,0,blend_radius_m)
    |   movel([0.171898, -1.383715, -2.567244, -0.761430, 1.570796, 1.742694],accel_mss,speed_ms,0,blend_radius_m)
    |   movel([0.172412, -1.383641, -2.567296, -0.761451, 1.570796, 1.743208],accel_mss,speed_ms,0,blend_radius_m)
    |   movel([0.172922, -1.383577, -2.567342, -0.761470, 1.570796, 1.743718],accel_mss,speed_ms,0,blend_radius_m)
    |   movel([0.173430, -1.383522, -2.567381, -0.761486, 1.570796, 1.744227],accel_mss,speed_ms,0,blend_radius_m)
    |   movel([0.173893, -1.383483, -2.567409, -0.761497, 1.570796, 1.744689],accel_mss,speed_ms,0,blend_radius_m)
    |   movel([0.174352, -1.383454, -2.567429, -0.761505, 1.570796, 1.745148],accel_mss,speed_ms,0,blend_radius_m)
    |   movel([0.174805, -1.383437, -2.567442, -0.761510, 1.570796, 1.745602],accel_mss,speed_ms,0,blend_radius_m)
    |   movel([0.175297, -1.383428, -2.567448, -0.761513, 1.570796, 1.746094],accel_mss,speed_ms,0,blend_radius_m)
    |   movel([0.175784, -1.383433, -2.567444, -0.761511, 1.570796, 1.746581],accel_mss,speed_ms,0,blend_radius_m)
    |   movel([0.176264, -1.383449, -2.567433, -0.761507, 1.570796, 1.747061],accel_mss,speed_ms,0,blend_radius_m)
    |   movel([0.176740, -1.383476, -2.567414, -0.761499, 1.570796, 1.747536],accel_mss,speed_ms,0,blend_radius_m)
    |   movel([0.177194, -1.383512, -2.567388, -0.761489, 1.570796, 1.747991],accel_mss,speed_ms,0,blend_radius_m)
    |   movel([0.177641, -1.383562, -2.567352, -0.761474, 1.570796, 1.748438],accel_mss,speed_ms,0,blend_radius_m)
    |   movel([0.178081, -1.383625, -2.567308, -0.761456, 1.570796, 1.748877],accel_mss,speed_ms,0,blend_radius_m)
    |   movel([0.178513, -1.383700, -2.567255, -0.761434, 1.570796, 1.749310],accel_mss,speed_ms,0,blend_radius_m)
    |   movel([0.178946, -1.383786, -2.567194, -0.761410, 1.570796, 1.749742],accel_mss,speed_ms,0,blend_radius_m)
    |   movel([0.179368, -1.383886, -2.567122, -0.761380, 1.570796, 1.750164],accel_mss,speed_ms,0,blend_radius_m)
    |   movel([0.179783, -1.383997, -2.567043, -0.761349, 1.570796, 1.750579],accel_mss,speed_ms,0,blend_radius_m)
    |   movel([0.180191, -1.384120, -2.566956, -0.761313, 1.570796, 1.750987],accel_mss,speed_ms,0,blend_radius_m)
    |   movel([0.180612, -1.384261, -2.566855, -0.761272, 1.570796, 1.751408],accel_mss,speed_ms,0,blend_radius_m)
    |   movel([0.181027, -1.384414, -2.566746, -0.761228, 1.570796, 1.751824],accel_mss,speed_ms,0,blend_radius_m)
    |   movel([0.181434, -1.384576, -2.566631, -0.761182, 1.570796, 1.752230],accel_mss,speed_ms,0,blend_radius_m)
    |   movel([0.181831, -1.384748, -2.566509, -0.761132, 1.570796, 1.752627],accel_mss,speed_ms,0,blend_radius_m)
    |   movel([0.183068, -1.385310, -2.566108, -0.760971, 1.570796, 1.753865],accel_mss,speed_ms,0,blend_radius_m)
    |   movel([0.210273, -1.379970, -2.569896, -0.762523, 1.570796, 1.781069],accel_mss,speed_ms,0,blend_radius_m)
    |   movel([0.237482, -1.375207, -2.573241, -0.763941, 1.570796, 1.808279],accel_mss,speed_ms,0,blend_radius_m)
    |   movel([0.237078, -1.376744, -2.572166, -0.763480, 1.570796, 1.807874],accel_mss,speed_ms,0,blend_radius_m)
    |   movel([0.236835, -1.377713, -2.571485, -0.763191, 1.570796, 1.807631],accel_mss,speed_ms,0,blend_radius_m)
    |   movel([0.236802, -1.377899, -2.571355, -0.763135, 1.570796, 1.807599],accel_mss,speed_ms,0,blend_radius_m)
    |   movel([0.236795, -1.378079, -2.571228, -0.763082, 1.570796, 1.807591],accel_mss,speed_ms,0,blend_radius_m)
    |   movel([0.236819, -1.378184, -2.571154, -0.763051, 1.570796, 1.807615],accel_mss,speed_ms,0,blend_radius_m)
    |   movel([0.236885, -1.378262, -2.571100, -0.763028, 1.570796, 1.807681],accel_mss,speed_ms,0,blend_radius_m)
    |   movel([0.236998, -1.378329, -2.571052, -0.763008, 1.570796, 1.807794],accel_mss,speed_ms,0,blend_radius_m)
    |   movel([0.237133, -1.378370, -2.571024, -0.762996, 1.570796, 1.807929],accel_mss,speed_ms,0,blend_radius_m)
    |   movel([0.237340, -1.378392, -2.571008, -0.762989, 1.570796, 1.808136],accel_mss,speed_ms,0,blend_radius_m)
    |   movel([0.237564, -1.378377, -2.571019, -0.762993, 1.570796, 1.808360],accel_mss,speed_ms,0,blend_radius_m)
    |   movel([0.246712, -1.377002, -2.571984, -0.763403, 1.570796, 1.817508],accel_mss,speed_ms,0,blend_radius_m)
    |   movel([0.253311, -1.376006, -2.572682, -0.763701, 1.570796, 1.824108],accel_mss,speed_ms,0,blend_radius_m)
    |   movel([0.269013, -1.373753, -2.574255, -0.764381, 1.570796, 1.839809],accel_mss,speed_ms,0,blend_radius_m)
    |   movel([0.269859, -1.370897, -2.576240, -0.765253, 1.570796, 1.840655],accel_mss,speed_ms,0,blend_radius_m)
    |   movel([0.270096, -1.370112, -2.576782, -0.765494, 1.570796, 1.840892],accel_mss,speed_ms,0,blend_radius_m)
    |   movel([0.270336, -1.369327, -2.577325, -0.765737, 1.570796, 1.841132],accel_mss,speed_ms,0,blend_radius_m)
    |   movel([0.270474, -1.368908, -2.577614, -0.765867, 1.570796, 1.841271],accel_mss,speed_ms,0,blend_radius_m)
    |   movel([0.270632, -1.368489, -2.577903, -0.765997, 1.570796, 1.841428],accel_mss,speed_ms,0,blend_radius_m)
    |   movel([0.270704, -1.368316, -2.578022, -0.766051, 1.570796, 1.841501],accel_mss,speed_ms,0,blend_radius_m)
    |   movel([0.270783, -1.368144, -2.578141, -0.766104, 1.570796, 1.841580],accel_mss,speed_ms,0,blend_radius_m)
    |   movel([0.270875, -1.367971, -2.578260, -0.766158, 1.570796, 1.841671],accel_mss,speed_ms,0,blend_radius_m)
    |   movel([0.270926, -1.367885, -2.578319, -0.766185, 1.570796, 1.841723],accel_mss,speed_ms,0,blend_radius_m)
    |   movel([0.270989, -1.367801, -2.578377, -0.766211, 1.570796, 1.841785],accel_mss,speed_ms,0,blend_radius_m)
    |   movel([0.271057, -1.367724, -2.578430, -0.766235, 1.570796, 1.841853],accel_mss,speed_ms,0,blend_radius_m)
    |   movel([0.271136, -1.367647, -2.578483, -0.766259, 1.570796, 1.841932],accel_mss,speed_ms,0,blend_radius_m)
    |   movel([0.271245, -1.367559, -2.578543, -0.766286, 1.570796, 1.842041],accel_mss,speed_ms,0,blend_radius_m)
    |   movel([0.271361, -1.367484, -2.578595, -0.766310, 1.570796, 1.842158],accel_mss,speed_ms,0,blend_radius_m)
    |   movel([0.271483, -1.367423, -2.578637, -0.766329, 1.570796, 1.842279],accel_mss,speed_ms,0,blend_radius_m)
    |   movel([0.271607, -1.367377, -2.578669, -0.766343, 1.570796, 1.842404],accel_mss,speed_ms,0,blend_radius_m)
    |   movel([0.271728, -1.367350, -2.578688, -0.766352, 1.570796, 1.842525],accel_mss,speed_ms,0,blend_radius_m)
    |   movel([0.273500, -1.367072, -2.578878, -0.766439, 1.570796, 1.844296],accel_mss,speed_ms,0,blend_radius_m)
    |   movel([0.275268, -1.366808, -2.579060, -0.766521, 1.570796, 1.846064],accel_mss,speed_ms,0,blend_radius_m)
    |   movel([0.278327, -1.366372, -2.579359, -0.766658, 1.570796, 1.849124],accel_mss,speed_ms,0,blend_radius_m)
    |   movel([0.281378, -1.365961, -2.579641, -0.766787, 1.570796, 1.852174],accel_mss,speed_ms,0,blend_radius_m)
    |   movel([0.298399, -1.363872, -2.581070, -0.767447, 1.570796, 1.869196],accel_mss,speed_ms,0,blend_radius_m)
    |   movel([0.325115, -1.361107, -2.582953, -0.768329, 1.570796, 1.895911],accel_mss,speed_ms,0,blend_radius_m)
    |   movel([0.326091, -1.358333, -2.584831, -0.769226, 1.570796, 1.896887],accel_mss,speed_ms,0,blend_radius_m)
    |   movel([0.327073, -1.355546, -2.586706, -0.770137, 1.570796, 1.897869],accel_mss,speed_ms,0,blend_radius_m)
    |   movel([0.310855, -1.352400, -2.588810, -0.771179, 1.570796, 1.881651],accel_mss,speed_ms,0,blend_radius_m)
    |   movel([0.294388, -1.349599, -2.590672, -0.772118, 1.570796, 1.865184],accel_mss,speed_ms,0,blend_radius_m)
    |   movel([0.294330, -1.349622, -2.590657, -0.772110, 1.570796, 1.865126],accel_mss,speed_ms,0,blend_radius_m)
    |   movel([0.294286, -1.349678, -2.590620, -0.772091, 1.570796, 1.865082],accel_mss,speed_ms,0,blend_radius_m)
    |   movel([0.292330, -1.353050, -2.588377, -0.770962, 1.570796, 1.863126],accel_mss,speed_ms,0,blend_radius_m)
    |   movel([0.286074, -1.354964, -2.587097, -0.770329, 1.570796, 1.856871],accel_mss,speed_ms,0,blend_radius_m)
    |   movel([0.283659, -1.355706, -2.586599, -0.770084, 1.570796, 1.854455],accel_mss,speed_ms,0,blend_radius_m)
    |   movel([0.281574, -1.356341, -2.586172, -0.769876, 1.570796, 1.852370],accel_mss,speed_ms,0,blend_radius_m)
    |   movel([0.279765, -1.356889, -2.585803, -0.769696, 1.570796, 1.850561],accel_mss,speed_ms,0,blend_radius_m)
    |   movel([0.279641, -1.356922, -2.585782, -0.769686, 1.570796, 1.850437],accel_mss,speed_ms,0,blend_radius_m)
    |   movel([0.279523, -1.356942, -2.585768, -0.769679, 1.570796, 1.850319],accel_mss,speed_ms,0,blend_radius_m)
    |   movel([0.279396, -1.356950, -2.585762, -0.769676, 1.570796, 1.850193],accel_mss,speed_ms,0,blend_radius_m)
    |   movel([0.279278, -1.356942, -2.585768, -0.769679, 1.570796, 1.850074],accel_mss,speed_ms,0,blend_radius_m)
    |   movel([0.279168, -1.356918, -2.585784, -0.769687, 1.570796, 1.849965],accel_mss,speed_ms,0,blend_radius_m)
    |   movel([0.270327, -1.354216, -2.587597, -0.770576, 1.570796, 1.841124],accel_mss,speed_ms,0,blend_radius_m)
    |   movel([0.261415, -1.351607, -2.589338, -0.771443, 1.570796, 1.832211],accel_mss,speed_ms,0,blend_radius_m)
    |   movel([0.261302, -1.351566, -2.589366, -0.771457, 1.570796, 1.832098],accel_mss,speed_ms,0,blend_radius_m)
    |   movel([0.261203, -1.351510, -2.589403, -0.771476, 1.570796, 1.831999],accel_mss,speed_ms,0,blend_radius_m)
    |   movel([0.261118, -1.351438, -2.589451, -0.771500, 1.570796, 1.831914],accel_mss,speed_ms,0,blend_radius_m)
    |   movel([0.261097, -1.351400, -2.589476, -0.771513, 1.570796, 1.831893],accel_mss,speed_ms,0,blend_radius_m)
    |   movel([0.261096, -1.351353, -2.589507, -0.771528, 1.570796, 1.831892],accel_mss,speed_ms,0,blend_radius_m)
    |   movel([0.261113, -1.351301, -2.589542, -0.771546, 1.570796, 1.831910],accel_mss,speed_ms,0,blend_radius_m)
    |   movel([0.263957, -1.345753, -2.593211, -0.773425, 1.570796, 1.834753],accel_mss,speed_ms,0,blend_radius_m)
    |   movel([0.266811, -1.340203, -2.596839, -0.775347, 1.570796, 1.837608],accel_mss,speed_ms,0,blend_radius_m)
    |   movel([0.266866, -1.340115, -2.596896, -0.775378, 1.570796, 1.837662],accel_mss,speed_ms,0,blend_radius_m)
    |   movel([0.266935, -1.340029, -2.596952, -0.775408, 1.570796, 1.837731],accel_mss,speed_ms,0,blend_radius_m)
    |   movel([0.267016, -1.339950, -2.597004, -0.775436, 1.570796, 1.837812],accel_mss,speed_ms,0,blend_radius_m)
    |   movel([0.267045, -1.339932, -2.597016, -0.775442, 1.570796, 1.837842],accel_mss,speed_ms,0,blend_radius_m)
    |   movel([0.267077, -1.339922, -2.597022, -0.775445, 1.570796, 1.837874],accel_mss,speed_ms,0,blend_radius_m)
    |   movel([0.267102, -1.339927, -2.597018, -0.775443, 1.570796, 1.837899],accel_mss,speed_ms,0,blend_radius_m)
    |   movel([0.268725, -1.340685, -2.596525, -0.775178, 1.570796, 1.839521],accel_mss,speed_ms,0,blend_radius_m)
    |   movel([0.269631, -1.341116, -2.596245, -0.775028, 1.570796, 1.840427],accel_mss,speed_ms,0,blend_radius_m)
    |   movel([0.270532, -1.341553, -2.595961, -0.774875, 1.570796, 1.841328],accel_mss,speed_ms,0,blend_radius_m)
    |   movel([0.272650, -1.342607, -2.595273, -0.774509, 1.570796, 1.843446],accel_mss,speed_ms,0,blend_radius_m)
    |   movel([0.278166, -1.345346, -2.593479, -0.773564, 1.570796, 1.848963],accel_mss,speed_ms,0,blend_radius_m)
    |   movel([0.278285, -1.345202, -2.593573, -0.773614, 1.570796, 1.849081],accel_mss,speed_ms,0,blend_radius_m)
    |   movel([0.278376, -1.345050, -2.593673, -0.773666, 1.570796, 1.849173],accel_mss,speed_ms,0,blend_radius_m)
    |   movel([0.283830, -1.334080, -2.600793, -0.777516, 1.570796, 1.854627],accel_mss,speed_ms,0,blend_radius_m)
    |   movel([0.283836, -1.333973, -2.600862, -0.777555, 1.570796, 1.854633],accel_mss,speed_ms,0,blend_radius_m)
    |   movel([0.283822, -1.333940, -2.600883, -0.777566, 1.570796, 1.854618],accel_mss,speed_ms,0,blend_radius_m)
    |   movel([0.283787, -1.333927, -2.600891, -0.777571, 1.570796, 1.854584],accel_mss,speed_ms,0,blend_radius_m)
    |   movel([0.283742, -1.333931, -2.600889, -0.777570, 1.570796, 1.854539],accel_mss,speed_ms,0,blend_radius_m)
    |   movel([0.278636, -1.335522, -2.599867, -0.777001, 1.570796, 1.849432],accel_mss,speed_ms,0,blend_radius_m)
    |   movel([0.275412, -1.336580, -2.599185, -0.776624, 1.570796, 1.846208],accel_mss,speed_ms,0,blend_radius_m)
    |   movel([0.272189, -1.337651, -2.598493, -0.776245, 1.570796, 1.842985],accel_mss,speed_ms,0,blend_radius_m)
    |   movel([0.270827, -1.338099, -2.598203, -0.776086, 1.570796, 1.841623],accel_mss,speed_ms,0,blend_radius_m)
    |   movel([0.269467, -1.338543, -2.597916, -0.775930, 1.570796, 1.840264],accel_mss,speed_ms,0,blend_radius_m)
    |   movel([0.267045, -1.339332, -2.597405, -0.775652, 1.570796, 1.837841],accel_mss,speed_ms,0,blend_radius_m)
    |   movel([0.267009, -1.339338, -2.597401, -0.775650, 1.570796, 1.837805],accel_mss,speed_ms,0,blend_radius_m)
    |   movel([0.266979, -1.339333, -2.597404, -0.775652, 1.570796, 1.837775],accel_mss,speed_ms,0,blend_radius_m)
    |   movel([0.266956, -1.339318, -2.597413, -0.775657, 1.570796, 1.837753],accel_mss,speed_ms,0,blend_radius_m)
    |   movel([0.266937, -1.339285, -2.597435, -0.775669, 1.570796, 1.837733],accel_mss,speed_ms,0,blend_radius_m)
    |   movel([0.266937, -1.339241, -2.597464, -0.775684, 1.570796, 1.837734],accel_mss,speed_ms,0,blend_radius_m)
    |   movel([0.266954, -1.339193, -2.597495, -0.775701, 1.570796, 1.837750],accel_mss,speed_ms,0,blend_radius_m)
    |   movel([0.269758, -1.333828, -2.600955, -0.777606, 1.570796, 1.840554],accel_mss,speed_ms,0,blend_radius_m)
    |   movel([0.272554, -1.328496, -2.604354, -0.779539, 1.570796, 1.843350],accel_mss,speed_ms,0,blend_radius_m)
    |   movel([0.272617, -1.328389, -2.604422, -0.779578, 1.570796, 1.843414],accel_mss,speed_ms,0,blend_radius_m)
    |   movel([0.272695, -1.328283, -2.604489, -0.779617, 1.570796, 1.843491],accel_mss,speed_ms,0,blend_radius_m)
    |   movel([0.272783, -1.328186, -2.604551, -0.779652, 1.570796, 1.843579],accel_mss,speed_ms,0,blend_radius_m)
    |   movel([0.272808, -1.328165, -2.604564, -0.779660, 1.570796, 1.843605],accel_mss,speed_ms,0,blend_radius_m)
    |   movel([0.272831, -1.328155, -2.604570, -0.779664, 1.570796, 1.843627],accel_mss,speed_ms,0,blend_radius_m)
    |   movel([0.277063, -1.326669, -2.605510, -0.780209, 1.570796, 1.847860],accel_mss,speed_ms,0,blend_radius_m)
    |   movel([0.281743, -1.325045, -2.606534, -0.780810, 1.570796, 1.852540],accel_mss,speed_ms,0,blend_radius_m)
    |   movel([0.287304, -1.323139, -2.607732, -0.781519, 1.570796, 1.858101],accel_mss,speed_ms,0,blend_radius_m)
    |   movel([0.301842, -1.318261, -2.610774, -0.783355, 1.570796, 1.872638],accel_mss,speed_ms,0,blend_radius_m)
    |   movel([0.305000, -1.322096, -2.608385, -0.781908, 1.570796, 1.875797],accel_mss,speed_ms,0,blend_radius_m)
    |   movel([0.308129, -1.325929, -2.605977, -0.780483, 1.570796, 1.878925],accel_mss,speed_ms,0,blend_radius_m)
    |   movel([0.307107, -1.327688, -2.604866, -0.779835, 1.570796, 1.877903],accel_mss,speed_ms,0,blend_radius_m)
    |   movel([0.306721, -1.328369, -2.604435, -0.779585, 1.570796, 1.877518],accel_mss,speed_ms,0,blend_radius_m)
    |   movel([0.306411, -1.328958, -2.604061, -0.779370, 1.570796, 1.877207],accel_mss,speed_ms,0,blend_radius_m)
    |   movel([0.306157, -1.329502, -2.603716, -0.779171, 1.570796, 1.876953],accel_mss,speed_ms,0,blend_radius_m)
    |   movel([0.306172, -1.329545, -2.603689, -0.779156, 1.570796, 1.876968],accel_mss,speed_ms,0,blend_radius_m)
    |   movel([0.306268, -1.329624, -2.603638, -0.779127, 1.570796, 1.877064],accel_mss,speed_ms,0,blend_radius_m)
    |   movel([0.306398, -1.329664, -2.603613, -0.779112, 1.570796, 1.877195],accel_mss,speed_ms,0,blend_radius_m)
    |   movel([0.311213, -1.330285, -2.603218, -0.778886, 1.570796, 1.882010],accel_mss,speed_ms,0,blend_radius_m)
    |   movel([0.320437, -1.331460, -2.602469, -0.778460, 1.570796, 1.891234],accel_mss,speed_ms,0,blend_radius_m)
    |   movel([0.323558, -1.331893, -2.602193, -0.778303, 1.570796, 1.894354],accel_mss,speed_ms,0,blend_radius_m)
    |   movel([0.324925, -1.332093, -2.602065, -0.778231, 1.570796, 1.895722],accel_mss,speed_ms,0,blend_radius_m)
    |   movel([0.326283, -1.332305, -2.601929, -0.778154, 1.570796, 1.897079],accel_mss,speed_ms,0,blend_radius_m)
    |   movel([0.327633, -1.332530, -2.601786, -0.778073, 1.570796, 1.898430],accel_mss,speed_ms,0,blend_radius_m)
    |   movel([0.328698, -1.332718, -2.601666, -0.778006, 1.570796, 1.899494],accel_mss,speed_ms,0,blend_radius_m)
    |   movel([0.329757, -1.332919, -2.601537, -0.777933, 1.570796, 1.900553],accel_mss,speed_ms,0,blend_radius_m)
    |   movel([0.330806, -1.333131, -2.601401, -0.777857, 1.570796, 1.901602],accel_mss,speed_ms,0,blend_radius_m)
    |   movel([0.331849, -1.333355, -2.601258, -0.777776, 1.570796, 1.902645],accel_mss,speed_ms,0,blend_radius_m)
    |   movel([0.332884, -1.333590, -2.601107, -0.777692, 1.570796, 1.903680],accel_mss,speed_ms,0,blend_radius_m)
    |   movel([0.333909, -1.333839, -2.600947, -0.777602, 1.570796, 1.904705],accel_mss,speed_ms,0,blend_radius_m)
    |   movel([0.334919, -1.334100, -2.600780, -0.777509, 1.570796, 1.905716],accel_mss,speed_ms,0,blend_radius_m)
    |   movel([0.335918, -1.334377, -2.600602, -0.777410, 1.570796, 1.906715],accel_mss,speed_ms,0,blend_radius_m)
    |   movel([0.336903, -1.334674, -2.600412, -0.777304, 1.570796, 1.907699],accel_mss,speed_ms,0,blend_radius_m)
    |   movel([0.337876, -1.334983, -2.600213, -0.777193, 1.570796, 1.908673],accel_mss,speed_ms,0,blend_radius_m)
    |   movel([0.338838, -1.335312, -2.600002, -0.777076, 1.570796, 1.909634],accel_mss,speed_ms,0,blend_radius_m)
    |   movel([0.339784, -1.335659, -2.599778, -0.776952, 1.570796, 1.910581],accel_mss,speed_ms,0,blend_radius_m)
    |   movel([0.340718, -1.336020, -2.599545, -0.776823, 1.570796, 1.911514],accel_mss,speed_ms,0,blend_radius_m)
    |   movel([0.341639, -1.336400, -2.599301, -0.776688, 1.570796, 1.912435],accel_mss,speed_ms,0,blend_radius_m)
    |   movel([0.342213, -1.336651, -2.599139, -0.776599, 1.570796, 1.913009],accel_mss,speed_ms,0,blend_radius_m)
    |   movel([0.342773, -1.336920, -2.598966, -0.776504, 1.570796, 1.913569],accel_mss,speed_ms,0,blend_radius_m)
    |   movel([0.343317, -1.337204, -2.598782, -0.776403, 1.570796, 1.914114],accel_mss,speed_ms,0,blend_radius_m)
    |   movel([0.343851, -1.337504, -2.598588, -0.776297, 1.570796, 1.914647],accel_mss,speed_ms,0,blend_radius_m)
    |   movel([0.344371, -1.337819, -2.598384, -0.776185, 1.570796, 1.915167],accel_mss,speed_ms,0,blend_radius_m)
    |   movel([0.344873, -1.338151, -2.598170, -0.776068, 1.570796, 1.915669],accel_mss,speed_ms,0,blend_radius_m)
    |   movel([0.345365, -1.338495, -2.597947, -0.775947, 1.570796, 1.916161],accel_mss,speed_ms,0,blend_radius_m)
    |   movel([0.345838, -1.338855, -2.597714, -0.775820, 1.570796, 1.916634],accel_mss,speed_ms,0,blend_radius_m)
    |   movel([0.346299, -1.339227, -2.597473, -0.775689, 1.570796, 1.917096],accel_mss,speed_ms,0,blend_radius_m)
    |   movel([0.346745, -1.339616, -2.597221, -0.775553, 1.570796, 1.917541],accel_mss,speed_ms,0,blend_radius_m)
    |   movel([0.347102, -1.339955, -2.597000, -0.775434, 1.570796, 1.917898],accel_mss,speed_ms,0,blend_radius_m)
    |   movel([0.347445, -1.340307, -2.596772, -0.775310, 1.570796, 1.918241],accel_mss,speed_ms,0,blend_radius_m)
    |   movel([0.347770, -1.340672, -2.596534, -0.775183, 1.570796, 1.918566],accel_mss,speed_ms,0,blend_radius_m)
    |   movel([0.348077, -1.341053, -2.596286, -0.775050, 1.570796, 1.918874],accel_mss,speed_ms,0,blend_radius_m)
    |   movel([0.348370, -1.341447, -2.596030, -0.774912, 1.570796, 1.919166],accel_mss,speed_ms,0,blend_radius_m)
    |   movel([0.348643, -1.341854, -2.595765, -0.774771, 1.570796, 1.919439],accel_mss,speed_ms,0,blend_radius_m)
    |   movel([0.348899, -1.342273, -2.595491, -0.774625, 1.570796, 1.919695],accel_mss,speed_ms,0,blend_radius_m)
    |   movel([0.349139, -1.342704, -2.595210, -0.774476, 1.570796, 1.919935],accel_mss,speed_ms,0,blend_radius_m)
    |   movel([0.349359, -1.343147, -2.594920, -0.774322, 1.570796, 1.920155],accel_mss,speed_ms,0,blend_radius_m)
    |   movel([0.349562, -1.343603, -2.594621, -0.774164, 1.570796, 1.920358],accel_mss,speed_ms,0,blend_radius_m)
    |   movel([0.349722, -1.344002, -2.594360, -0.774027, 1.570796, 1.920518],accel_mss,speed_ms,0,blend_radius_m)
    |   movel([0.349862, -1.344414, -2.594091, -0.773885, 1.570796, 1.920658],accel_mss,speed_ms,0,blend_radius_m)
    |   movel([0.349985, -1.344831, -2.593817, -0.773741, 1.570796, 1.920782],accel_mss,speed_ms,0,blend_radius_m)
    |   movel([0.350092, -1.345261, -2.593534, -0.773593, 1.570796, 1.920888],accel_mss,speed_ms,0,blend_radius_m)
    |   movel([0.350181, -1.345699, -2.593246, -0.773443, 1.570796, 1.920978],accel_mss,speed_ms,0,blend_radius_m)
    |   movel([0.350254, -1.346143, -2.592955, -0.773291, 1.570796, 1.921050],accel_mss,speed_ms,0,blend_radius_m)
    |   movel([0.350308, -1.346598, -2.592655, -0.773136, 1.570796, 1.921104],accel_mss,speed_ms,0,blend_radius_m)
    |   movel([0.350344, -1.347060, -2.592351, -0.772978, 1.570796, 1.921141],accel_mss,speed_ms,0,blend_radius_m)
    |   movel([0.350367, -1.347528, -2.592042, -0.772819, 1.570796, 1.921163],accel_mss,speed_ms,0,blend_radius_m)
    |   movel([0.350368, -1.348001, -2.591729, -0.772658, 1.570796, 1.921164],accel_mss,speed_ms,0,blend_radius_m)
    |   movel([0.350354, -1.348483, -2.591411, -0.772495, 1.570796, 1.921150],accel_mss,speed_ms,0,blend_radius_m)
    |   movel([0.350332, -1.348816, -2.591191, -0.772382, 1.570796, 1.921128],accel_mss,speed_ms,0,blend_radius_m)
    |   movel([0.350291, -1.349153, -2.590968, -0.772268, 1.570796, 1.921087],accel_mss,speed_ms,0,blend_radius_m)
    |   movel([0.350237, -1.349493, -2.590743, -0.772154, 1.570796, 1.921033],accel_mss,speed_ms,0,blend_radius_m)
    |   movel([0.350168, -1.349836, -2.590515, -0.772038, 1.570796, 1.920964],accel_mss,speed_ms,0,blend_radius_m)
    |   movel([0.350080, -1.350185, -2.590283, -0.771920, 1.570796, 1.920876],accel_mss,speed_ms,0,blend_radius_m)
    |   movel([0.349913, -1.350787, -2.589884, -0.771718, 1.570796, 1.920710],accel_mss,speed_ms,0,blend_radius_m)
    |   movel([0.349733, -1.351394, -2.589480, -0.771515, 1.570796, 1.920530],accel_mss,speed_ms,0,blend_radius_m)
    |   movel([0.349542, -1.351999, -2.589077, -0.771312, 1.570796, 1.920338],accel_mss,speed_ms,0,blend_radius_m)
    |   movel([0.349336, -1.352607, -2.588672, -0.771110, 1.570796, 1.920132],accel_mss,speed_ms,0,blend_radius_m)
    |   movel([0.349114, -1.353232, -2.588255, -0.770902, 1.570796, 1.919910],accel_mss,speed_ms,0,blend_radius_m)
    |   movel([0.348880, -1.353854, -2.587839, -0.770695, 1.570796, 1.919677],accel_mss,speed_ms,0,blend_radius_m)
    |   movel([0.348632, -1.354480, -2.587421, -0.770489, 1.570796, 1.919429],accel_mss,speed_ms,0,blend_radius_m)
    |   movel([0.348373, -1.355103, -2.587003, -0.770283, 1.570796, 1.919169],accel_mss,speed_ms,0,blend_radius_m)
    |   movel([0.348196, -1.355501, -2.586736, -0.770152, 1.570796, 1.918992],accel_mss,speed_ms,0,blend_radius_m)
    |   movel([0.348009, -1.355898, -2.586470, -0.770021, 1.570796, 1.918806],accel_mss,speed_ms,0,blend_radius_m)
    |   movel([0.347809, -1.356296, -2.586203, -0.769891, 1.570796, 1.918605],accel_mss,speed_ms,0,blend_radius_m)
    |   movel([0.347597, -1.356691, -2.585936, -0.769761, 1.570796, 1.918394],accel_mss,speed_ms,0,blend_radius_m)
    |   movel([0.347375, -1.357085, -2.585671, -0.769632, 1.570796, 1.918171],accel_mss,speed_ms,0,blend_radius_m)
    |   movel([0.347099, -1.357552, -2.585357, -0.769480, 1.570796, 1.917895],accel_mss,speed_ms,0,blend_radius_m)
    |   movel([0.346814, -1.358018, -2.585043, -0.769328, 1.570796, 1.917610],accel_mss,speed_ms,0,blend_radius_m)
    |   movel([0.346707, -1.358186, -2.584929, -0.769273, 1.570796, 1.917503],accel_mss,speed_ms,0,blend_radius_m)
    |   movel([0.346590, -1.358348, -2.584820, -0.769221, 1.570796, 1.917386],accel_mss,speed_ms,0,blend_radius_m)
    |   movel([0.346461, -1.358510, -2.584711, -0.769168, 1.570796, 1.917257],accel_mss,speed_ms,0,blend_radius_m)
    |   movel([0.346356, -1.358628, -2.584631, -0.769130, 1.570796, 1.917152],accel_mss,speed_ms,0,blend_radius_m)
    |   movel([0.346242, -1.358739, -2.584556, -0.769094, 1.570796, 1.917038],accel_mss,speed_ms,0,blend_radius_m)
    |   movel([0.346118, -1.358844, -2.584485, -0.769060, 1.570796, 1.916914],accel_mss,speed_ms,0,blend_radius_m)
    |   movel([0.345968, -1.358955, -2.584410, -0.769024, 1.570796, 1.916764],accel_mss,speed_ms,0,blend_radius_m)
    |   movel([0.345813, -1.359060, -2.584339, -0.768990, 1.570796, 1.916610],accel_mss,speed_ms,0,blend_radius_m)
    |   movel([0.345658, -1.359156, -2.584275, -0.768959, 1.570796, 1.916454],accel_mss,speed_ms,0,blend_radius_m)
    |   movel([0.345229, -1.359415, -2.584099, -0.768875, 1.570796, 1.916025],accel_mss,speed_ms,0,blend_radius_m)
    |   movel([0.345135, -1.359484, -2.584053, -0.768852, 1.570796, 1.915932],accel_mss,speed_ms,0,blend_radius_m)
    |   movel([0.345053, -1.359565, -2.583998, -0.768826, 1.570796, 1.915850],accel_mss,speed_ms,0,blend_radius_m)
    |   movel([0.345015, -1.359630, -2.583954, -0.768805, 1.570796, 1.915811],accel_mss,speed_ms,0,blend_radius_m)
    |   movel([0.345009, -1.359689, -2.583914, -0.768786, 1.570796, 1.915806],accel_mss,speed_ms,0,blend_radius_m)
    |   movel([0.345082, -1.359818, -2.583826, -0.768744, 1.570796, 1.915878],accel_mss,speed_ms,0,blend_radius_m)
    |   movel([0.345117, -1.359868, -2.583793, -0.768728, 1.570796, 1.915914],accel_mss,speed_ms,0,blend_radius_m)
    |   movel([0.345141, -1.359926, -2.583754, -0.768710, 1.570796, 1.915937],accel_mss,speed_ms,0,blend_radius_m)
    |   movel([0.345151, -1.359993, -2.583708, -0.768688, 1.570796, 1.915947],accel_mss,speed_ms,0,blend_radius_m)
    |   movel([0.345146, -1.360064, -2.583660, -0.768665, 1.570796, 1.915942],accel_mss,speed_ms,0,blend_radius_m)
    |   movel([0.345127, -1.360138, -2.583609, -0.768641, 1.570796, 1.915924],accel_mss,speed_ms,0,blend_radius_m)
    |   movel([0.344852, -1.360980, -2.583039, -0.768370, 1.570796, 1.915649],accel_mss,speed_ms,0,blend_radius_m)
    |   movel([0.344566, -1.361822, -2.582467, -0.768100, 1.570796, 1.915362],accel_mss,speed_ms,0,blend_radius_m)
    |   movel([0.344087, -1.363189, -2.581536, -0.767664, 1.570796, 1.914883],accel_mss,speed_ms,0,blend_radius_m)
    |   movel([0.343595, -1.364554, -2.580604, -0.767231, 1.570796, 1.914391],accel_mss,speed_ms,0,blend_radius_m)
    |   movel([0.341468, -1.370323, -2.576637, -0.765429, 1.570796, 1.912264],accel_mss,speed_ms,0,blend_radius_m)
    |   movel([0.337741, -1.380449, -2.569558, -0.762382, 1.570796, 1.908537],accel_mss,speed_ms,0,blend_radius_m)
    |   movel([0.341498, -1.380139, -2.569777, -0.762473, 1.570796, 1.912294],accel_mss,speed_ms,0,blend_radius_m)
    |   movel([0.345249, -1.379843, -2.569986, -0.762560, 1.570796, 1.916046],accel_mss,speed_ms,0,blend_radius_m)
    |   movel([0.348358, -1.373140, -2.574682, -0.764567, 1.570796, 1.919155],accel_mss,speed_ms,0,blend_radius_m)
    |   movel([0.349582, -1.370513, -2.576506, -0.765371, 1.570796, 1.920378],accel_mss,speed_ms,0,blend_radius_m)
    |   movel([0.350659, -1.368204, -2.578099, -0.766085, 1.570796, 1.921455],accel_mss,speed_ms,0,blend_radius_m)
    |   movel([0.351587, -1.366221, -2.579462, -0.766705, 1.570796, 1.922383],accel_mss,speed_ms,0,blend_radius_m)
    |   movel([0.351778, -1.365822, -2.579736, -0.766831, 1.570796, 1.922574],accel_mss,speed_ms,0,blend_radius_m)
    |   movel([0.351845, -1.365700, -2.579820, -0.766869, 1.570796, 1.922642],accel_mss,speed_ms,0,blend_radius_m)
    |   movel([0.351926, -1.365579, -2.579903, -0.766907, 1.570796, 1.922723],accel_mss,speed_ms,0,blend_radius_m)
    |   movel([0.352026, -1.365453, -2.579989, -0.766947, 1.570796, 1.922822],accel_mss,speed_ms,0,blend_radius_m)
    |   movel([0.352139, -1.365327, -2.580075, -0.766986, 1.570796, 1.922935],accel_mss,speed_ms,0,blend_radius_m)
    |   movel([0.352259, -1.365209, -2.580157, -0.767024, 1.570796, 1.923055],accel_mss,speed_ms,0,blend_radius_m)
    |   movel([0.352388, -1.365096, -2.580234, -0.767059, 1.570796, 1.923184],accel_mss,speed_ms,0,blend_radius_m)
    |   movel([0.352517, -1.364997, -2.580301, -0.767091, 1.570796, 1.923313],accel_mss,speed_ms,0,blend_radius_m)
    |   movel([0.352648, -1.364909, -2.580361, -0.767118, 1.570796, 1.923445],accel_mss,speed_ms,0,blend_radius_m)
    |   movel([0.352779, -1.364837, -2.580411, -0.767141, 1.570796, 1.923575],accel_mss,speed_ms,0,blend_radius_m)
    |   movel([0.352912, -1.364776, -2.580452, -0.767160, 1.570796, 1.923708],accel_mss,speed_ms,0,blend_radius_m)
    |   movel([0.353044, -1.364729, -2.580484, -0.767175, 1.570796, 1.923841],accel_mss,speed_ms,0,blend_radius_m)
    |   movel([0.353176, -1.364698, -2.580506, -0.767185, 1.570796, 1.923972],accel_mss,speed_ms,0,blend_radius_m)
    |   movel([0.353419, -1.364656, -2.580535, -0.767198, 1.570796, 1.924215],accel_mss,speed_ms,0,blend_radius_m)
    |   movel([0.353654, -1.364629, -2.580553, -0.767207, 1.570796, 1.924450],accel_mss,speed_ms,0,blend_radius_m)
    |   movel([0.353886, -1.364617, -2.580561, -0.767211, 1.570796, 1.924682],accel_mss,speed_ms,0,blend_radius_m)
    |   movel([0.354305, -1.364609, -2.580567, -0.767213, 1.570796, 1.925102],accel_mss,speed_ms,0,blend_radius_m)
    |   movel([0.354722, -1.364610, -2.580566, -0.767213, 1.570796, 1.925518],accel_mss,speed_ms,0,blend_radius_m)
    |   movel([0.355132, -1.364621, -2.580559, -0.767210, 1.570796, 1.925928],accel_mss,speed_ms,0,blend_radius_m)
    |   movel([0.358511, -1.364757, -2.580465, -0.767166, 1.570796, 1.929307],accel_mss,speed_ms,0,blend_radius_m)
    |   movel([0.360563, -1.364852, -2.580400, -0.767136, 1.570796, 1.931360],accel_mss,speed_ms,0,blend_radius_m)
    |   movel([0.362381, -1.364949, -2.580334, -0.767106, 1.570796, 1.933177],accel_mss,speed_ms,0,blend_radius_m)
    |   movel([0.363914, -1.365036, -2.580274, -0.767078, 1.570796, 1.934710],accel_mss,speed_ms,0,blend_radius_m)
    |   movel([0.364121, -1.365050, -2.580265, -0.767074, 1.570796, 1.934918],accel_mss,speed_ms,0,blend_radius_m)
    |   movel([0.364326, -1.365071, -2.580250, -0.767067, 1.570796, 1.935122],accel_mss,speed_ms,0,blend_radius_m)
    |   movel([0.364488, -1.365099, -2.580231, -0.767058, 1.570796, 1.935284],accel_mss,speed_ms,0,blend_radius_m)
    |   movel([0.364643, -1.365139, -2.580204, -0.767046, 1.570796, 1.935440],accel_mss,speed_ms,0,blend_radius_m)
    |   movel([0.364791, -1.365193, -2.580167, -0.767029, 1.570796, 1.935587],accel_mss,speed_ms,0,blend_radius_m)
    |   movel([0.364874, -1.365236, -2.580138, -0.767015, 1.570796, 1.935670],accel_mss,speed_ms,0,blend_radius_m)
    |   movel([0.364948, -1.365291, -2.580100, -0.766998, 1.570796, 1.935745],accel_mss,speed_ms,0,blend_radius_m)
    |   movel([0.365012, -1.365354, -2.580057, -0.766978, 1.570796, 1.935809],accel_mss,speed_ms,0,blend_radius_m)
    |   movel([0.365066, -1.365426, -2.580007, -0.766955, 1.570796, 1.935862],accel_mss,speed_ms,0,blend_radius_m)
    |   movel([0.365106, -1.365502, -2.579956, -0.766931, 1.570796, 1.935903],accel_mss,speed_ms,0,blend_radius_m)
    |   movel([0.365132, -1.365585, -2.579899, -0.766905, 1.570796, 1.935929],accel_mss,speed_ms,0,blend_radius_m)
    |   movel([0.365148, -1.365675, -2.579837, -0.766877, 1.570796, 1.935945],accel_mss,speed_ms,0,blend_radius_m)
    |   movel([0.365152, -1.365768, -2.579773, -0.766848, 1.570796, 1.935948],accel_mss,speed_ms,0,blend_radius_m)
    |   movel([0.365136, -1.365915, -2.579673, -0.766802, 1.570796, 1.935932],accel_mss,speed_ms,0,blend_radius_m)
    |   movel([0.365103, -1.366064, -2.579570, -0.766755, 1.570796, 1.935899],accel_mss,speed_ms,0,blend_radius_m)
    |   movel([0.365051, -1.366215, -2.579467, -0.766707, 1.570796, 1.935847],accel_mss,speed_ms,0,blend_radius_m)
    |   movel([0.364962, -1.366506, -2.579267, -0.766616, 1.570796, 1.935759],accel_mss,speed_ms,0,blend_radius_m)
    |   movel([0.364956, -1.366593, -2.579208, -0.766589, 1.570796, 1.935753],accel_mss,speed_ms,0,blend_radius_m)
    |   movel([0.364981, -1.366666, -2.579157, -0.766566, 1.570796, 1.935778],accel_mss,speed_ms,0,blend_radius_m)
    |   movel([0.365038, -1.366725, -2.579117, -0.766547, 1.570796, 1.935834],accel_mss,speed_ms,0,blend_radius_m)
    |   movel([0.365115, -1.366759, -2.579093, -0.766536, 1.570796, 1.935911],accel_mss,speed_ms,0,blend_radius_m)
    |   movel([0.365424, -1.366812, -2.579057, -0.766520, 1.570796, 1.936220],accel_mss,speed_ms,0,blend_radius_m)
    |   movel([0.365730, -1.366846, -2.579034, -0.766509, 1.570796, 1.936526],accel_mss,speed_ms,0,blend_radius_m)
    |   movel([0.366203, -1.366895, -2.579000, -0.766494, 1.570796, 1.937000],accel_mss,speed_ms,0,blend_radius_m)
    |   movel([0.366739, -1.366952, -2.578961, -0.766476, 1.570796, 1.937535],accel_mss,speed_ms,0,blend_radius_m)
    |   movel([0.367259, -1.367010, -2.578921, -0.766458, 1.570796, 1.938056],accel_mss,speed_ms,0,blend_radius_m)
    |   movel([0.367921, -1.367089, -2.578867, -0.766433, 1.570796, 1.938717],accel_mss,speed_ms,0,blend_radius_m)
    |   movel([0.368574, -1.367185, -2.578801, -0.766403, 1.570796, 1.939370],accel_mss,speed_ms,0,blend_radius_m)
    |   movel([0.369216, -1.367295, -2.578725, -0.766369, 1.570796, 1.940012],accel_mss,speed_ms,0,blend_radius_m)
    |   movel([0.369849, -1.367423, -2.578637, -0.766329, 1.570796, 1.940645],accel_mss,speed_ms,0,blend_radius_m)
    |   movel([0.370471, -1.367564, -2.578540, -0.766285, 1.570796, 1.941267],accel_mss,speed_ms,0,blend_radius_m)
    |   movel([0.371085, -1.367721, -2.578432, -0.766236, 1.570796, 1.941881],accel_mss,speed_ms,0,blend_radius_m)
    |   movel([0.371688, -1.367891, -2.578315, -0.766183, 1.570796, 1.942485],accel_mss,speed_ms,0,blend_radius_m)
    |   movel([0.372280, -1.368079, -2.578186, -0.766124, 1.570796, 1.943076],accel_mss,speed_ms,0,blend_radius_m)
    |   movel([0.372862, -1.368279, -2.578048, -0.766062, 1.570796, 1.943658],accel_mss,speed_ms,0,blend_radius_m)
    |   movel([0.373430, -1.368495, -2.577899, -0.765995, 1.570796, 1.944226],accel_mss,speed_ms,0,blend_radius_m)
    |   movel([0.374070, -1.368761, -2.577715, -0.765912, 1.570796, 1.944867],accel_mss,speed_ms,0,blend_radius_m)
    |   movel([0.374700, -1.369042, -2.577522, -0.765825, 1.570796, 1.945496],accel_mss,speed_ms,0,blend_radius_m)
    |   movel([0.375312, -1.369342, -2.577315, -0.765732, 1.570796, 1.946109],accel_mss,speed_ms,0,blend_radius_m)
    |   movel([0.375911, -1.369657, -2.577097, -0.765635, 1.570796, 1.946708],accel_mss,speed_ms,0,blend_radius_m)
    |   movel([0.376496, -1.369988, -2.576868, -0.765532, 1.570796, 1.947292],accel_mss,speed_ms,0,blend_radius_m)
    |   movel([0.377065, -1.370334, -2.576629, -0.765426, 1.570796, 1.947861],accel_mss,speed_ms,0,blend_radius_m)
    |   movel([0.377619, -1.370699, -2.576376, -0.765313, 1.570796, 1.948415],accel_mss,speed_ms,0,blend_radius_m)
    |   movel([0.378158, -1.371077, -2.576115, -0.765197, 1.570796, 1.948955],accel_mss,speed_ms,0,blend_radius_m)
    |   movel([0.378681, -1.371470, -2.575842, -0.765077, 1.570796, 1.949477],accel_mss,speed_ms,0,blend_radius_m)
    |   movel([0.379194, -1.371885, -2.575554, -0.764949, 1.570796, 1.949990],accel_mss,speed_ms,0,blend_radius_m)
    |   movel([0.379692, -1.372315, -2.575256, -0.764818, 1.570796, 1.950488],accel_mss,speed_ms,0,blend_radius_m)
    |   movel([0.380172, -1.372758, -2.574948, -0.764683, 1.570796, 1.950968],accel_mss,speed_ms,0,blend_radius_m)
    |   movel([0.380636, -1.373216, -2.574629, -0.764544, 1.570796, 1.951432],accel_mss,speed_ms,0,blend_radius_m)
    |   movel([0.381084, -1.373688, -2.574300, -0.764400, 1.570796, 1.951881],accel_mss,speed_ms,0,blend_radius_m)
    |   movel([0.381515, -1.374175, -2.573962, -0.764253, 1.570796, 1.952311],accel_mss,speed_ms,0,blend_radius_m)
    |   movel([0.381927, -1.374675, -2.573612, -0.764102, 1.570796, 1.952724],accel_mss,speed_ms,0,blend_radius_m)
    |   movel([0.382323, -1.375187, -2.573255, -0.763947, 1.570796, 1.953119],accel_mss,speed_ms,0,blend_radius_m)
    |   movel([0.382700, -1.375714, -2.572887, -0.763789, 1.570796, 1.953497],accel_mss,speed_ms,0,blend_radius_m)
    |   movel([0.383056, -1.376247, -2.572513, -0.763628, 1.570796, 1.953852],accel_mss,speed_ms,0,blend_radius_m)
    |   movel([0.383395, -1.376793, -2.572131, -0.763465, 1.570796, 1.954191],accel_mss,speed_ms,0,blend_radius_m)
    |   movel([0.383715, -1.377352, -2.571739, -0.763298, 1.570796, 1.954512],accel_mss,speed_ms,0,blend_radius_m)
    |   movel([0.384015, -1.377923, -2.571338, -0.763128, 1.570796, 1.954811],accel_mss,speed_ms,0,blend_radius_m)
    |   movel([0.384298, -1.378503, -2.570930, -0.762956, 1.570796, 1.955094],accel_mss,speed_ms,0,blend_radius_m)
    |   movel([0.384564, -1.379097, -2.570512, -0.762780, 1.570796, 1.955360],accel_mss,speed_ms,0,blend_radius_m)
    |   movel([0.384808, -1.379702, -2.570085, -0.762601, 1.570796, 1.955604],accel_mss,speed_ms,0,blend_radius_m)
    |   movel([0.385034, -1.380317, -2.569652, -0.762420, 1.570796, 1.955830],accel_mss,speed_ms,0,blend_radius_m)
    |   movel([0.385241, -1.380943, -2.569209, -0.762237, 1.570796, 1.956038],accel_mss,speed_ms,0,blend_radius_m)
    |   movel([0.385413, -1.381515, -2.568804, -0.762069, 1.570796, 1.956209],accel_mss,speed_ms,0,blend_radius_m)
    |   movel([0.385569, -1.382095, -2.568394, -0.761900, 1.570796, 1.956366],accel_mss,speed_ms,0,blend_radius_m)
    |   movel([0.385709, -1.382681, -2.567979, -0.761730, 1.570796, 1.956505],accel_mss,speed_ms,0,blend_radius_m)
    |   movel([0.385833, -1.383276, -2.567556, -0.761557, 1.570796, 1.956629],accel_mss,speed_ms,0,blend_radius_m)
    |   movel([0.385943, -1.383877, -2.567129, -0.761383, 1.570796, 1.956739],accel_mss,speed_ms,0,blend_radius_m)
    |   movel([0.386039, -1.384483, -2.566697, -0.761208, 1.570796, 1.956835],accel_mss,speed_ms,0,blend_radius_m)
    |   movel([0.386119, -1.385098, -2.566259, -0.761032, 1.570796, 1.956915],accel_mss,speed_ms,0,blend_radius_m)
    |   movel([0.386198, -1.385864, -2.565713, -0.760812, 1.570796, 1.956994],accel_mss,speed_ms,0,blend_radius_m)
    |   movel([0.386259, -1.386639, -2.565159, -0.760591, 1.570796, 1.957055],accel_mss,speed_ms,0,blend_radius_m)
    |   movel([0.386300, -1.387418, -2.564602, -0.760370, 1.570796, 1.957096],accel_mss,speed_ms,0,blend_radius_m)
    |   movel([0.386325, -1.388205, -2.564037, -0.760147, 1.570796, 1.957122],accel_mss,speed_ms,0,blend_radius_m)
    |   movel([0.386330, -1.388996, -2.563469, -0.759924, 1.570796, 1.957127],accel_mss,speed_ms,0,blend_radius_m)
    |   movel([0.386319, -1.389793, -2.562896, -0.759700, 1.570796, 1.957115],accel_mss,speed_ms,0,blend_radius_m)
    |   movel([0.386287, -1.390579, -2.562330, -0.759480, 1.570796, 1.957083],accel_mss,speed_ms,0,blend_radius_m)
    |   movel([0.386239, -1.391369, -2.561760, -0.759260, 1.570796, 1.957035],accel_mss,speed_ms,0,blend_radius_m)
    |   movel([0.386173, -1.392162, -2.561187, -0.759040, 1.570796, 1.956970],accel_mss,speed_ms,0,blend_radius_m)
    |   movel([0.386087, -1.392962, -2.560608, -0.758819, 1.570796, 1.956883],accel_mss,speed_ms,0,blend_radius_m)
    |   movel([0.385985, -1.393765, -2.560026, -0.758598, 1.570796, 1.956781],accel_mss,speed_ms,0,blend_radius_m)
    |   movel([0.385864, -1.394570, -2.559441, -0.758377, 1.570796, 1.956660],accel_mss,speed_ms,0,blend_radius_m)
    |   movel([0.385758, -1.395194, -2.558988, -0.758207, 1.570796, 1.956554],accel_mss,speed_ms,0,blend_radius_m)
    |   movel([0.385635, -1.395819, -2.558533, -0.758037, 1.570796, 1.956431],accel_mss,speed_ms,0,blend_radius_m)
    |   movel([0.385494, -1.396448, -2.558074, -0.757867, 1.570796, 1.956290],accel_mss,speed_ms,0,blend_radius_m)
    |   movel([0.385339, -1.397079, -2.557613, -0.757696, 1.570796, 1.956135],accel_mss,speed_ms,0,blend_radius_m)
    |   movel([0.385167, -1.397713, -2.557151, -0.757526, 1.570796, 1.955963],accel_mss,speed_ms,0,blend_radius_m)
    |   movel([0.384980, -1.398345, -2.556688, -0.757356, 1.570796, 1.955776],accel_mss,speed_ms,0,blend_radius_m)
    |   movel([0.384777, -1.398982, -2.556221, -0.757186, 1.570796, 1.955573],accel_mss,speed_ms,0,blend_radius_m)
    |   movel([0.384630, -1.399460, -2.555871, -0.757059, 1.570796, 1.955426],accel_mss,speed_ms,0,blend_radius_m)
    |   movel([0.384503, -1.399937, -2.555521, -0.756932, 1.570796, 1.955299],accel_mss,speed_ms,0,blend_radius_m)
    |   movel([0.384489, -1.400035, -2.555448, -0.756906, 1.570796, 1.955285],accel_mss,speed_ms,0,blend_radius_m)
    |   movel([0.384501, -1.400125, -2.555382, -0.756882, 1.570796, 1.955297],accel_mss,speed_ms,0,blend_radius_m)
    |   movel([0.384534, -1.400203, -2.555325, -0.756861, 1.570796, 1.955330],accel_mss,speed_ms,0,blend_radius_m)
    |   movel([0.384586, -1.400265, -2.555279, -0.756845, 1.570796, 1.955383],accel_mss,speed_ms,0,blend_radius_m)
    |   movel([0.384697, -1.400340, -2.555224, -0.756825, 1.570796, 1.955494],accel_mss,speed_ms,0,blend_radius_m)
    |   movel([0.384829, -1.400392, -2.555186, -0.756811, 1.570796, 1.955625],accel_mss,speed_ms,0,blend_radius_m)
    |   movel([0.384977, -1.400420, -2.555165, -0.756804, 1.570796, 1.955773],accel_mss,speed_ms,0,blend_radius_m)
    |   movel([0.386589, -1.400548, -2.555071, -0.756770, 1.570796, 1.957385],accel_mss,speed_ms,0,blend_radius_m)
    |   movel([0.387961, -1.400643, -2.555002, -0.756745, 1.570796, 1.958758],accel_mss,speed_ms,0,blend_radius_m)
    |   movel([0.387632, -1.401194, -2.554596, -0.756599, 1.570796, 1.958429],accel_mss,speed_ms,0,blend_radius_m)
    |   movel([0.387398, -1.401608, -2.554291, -0.756490, 1.570796, 1.958194],accel_mss,speed_ms,0,blend_radius_m)
    |   movel([0.387179, -1.402022, -2.553986, -0.756381, 1.570796, 1.957975],accel_mss,speed_ms,0,blend_radius_m)
    |   movel([0.386433, -1.403535, -2.552868, -0.755986, 1.570796, 1.957229],accel_mss,speed_ms,0,blend_radius_m)
    |   movel([0.385609, -1.405284, -2.551572, -0.755533, 1.570796, 1.956406],accel_mss,speed_ms,0,blend_radius_m)
    |   movel([0.385590, -1.405417, -2.551473, -0.755499, 1.570796, 1.956386],accel_mss,speed_ms,0,blend_radius_m)
    |   movel([0.385602, -1.405467, -2.551436, -0.755486, 1.570796, 1.956399],accel_mss,speed_ms,0,blend_radius_m)
    |   movel([0.385637, -1.405501, -2.551411, -0.755477, 1.570796, 1.956434],accel_mss,speed_ms,0,blend_radius_m)
    |   movel([0.386465, -1.405895, -2.551118, -0.755376, 1.570796, 1.957261],accel_mss,speed_ms,0,blend_radius_m)
    |   movel([0.387009, -1.406109, -2.550959, -0.755321, 1.570796, 1.957805],accel_mss,speed_ms,0,blend_radius_m)
    |   movel([0.387430, -1.406275, -2.550836, -0.755278, 1.570796, 1.958226],accel_mss,speed_ms,0,blend_radius_m)
    |   movel([0.387838, -1.406454, -2.550702, -0.755233, 1.570796, 1.958634],accel_mss,speed_ms,0,blend_radius_m)
    |   movel([0.388233, -1.406647, -2.550559, -0.755183, 1.570796, 1.959030],accel_mss,speed_ms,0,blend_radius_m)
    |   movel([0.388618, -1.406855, -2.550404, -0.755130, 1.570796, 1.959414],accel_mss,speed_ms,0,blend_radius_m)
    |   movel([0.388990, -1.407076, -2.550239, -0.755074, 1.570796, 1.959786],accel_mss,speed_ms,0,blend_radius_m)
    |   movel([0.389347, -1.407311, -2.550064, -0.755014, 1.570796, 1.960143],accel_mss,speed_ms,0,blend_radius_m)
    |   movel([0.389707, -1.407570, -2.549871, -0.754948, 1.570796, 1.960503],accel_mss,speed_ms,0,blend_radius_m)
    |   movel([0.390054, -1.407837, -2.549672, -0.754880, 1.570796, 1.960851],accel_mss,speed_ms,0,blend_radius_m)
    |   movel([0.390386, -1.408120, -2.549460, -0.754808, 1.570796, 1.961182],accel_mss,speed_ms,0,blend_radius_m)
    |   movel([0.390707, -1.408412, -2.549243, -0.754734, 1.570796, 1.961503],accel_mss,speed_ms,0,blend_radius_m)
    |   movel([0.391015, -1.408717, -2.549015, -0.754657, 1.570796, 1.961811],accel_mss,speed_ms,0,blend_radius_m)
    |   movel([0.391310, -1.409031, -2.548780, -0.754578, 1.570796, 1.962107],accel_mss,speed_ms,0,blend_radius_m)
    |   movel([0.391597, -1.409364, -2.548531, -0.754494, 1.570796, 1.962394],accel_mss,speed_ms,0,blend_radius_m)
    |   movel([0.391868, -1.409708, -2.548273, -0.754408, 1.570796, 1.962664],accel_mss,speed_ms,0,blend_radius_m)
    |   movel([0.392127, -1.410064, -2.548007, -0.754319, 1.570796, 1.962923],accel_mss,speed_ms,0,blend_radius_m)
    |   movel([0.392371, -1.410427, -2.547734, -0.754227, 1.570796, 1.963167],accel_mss,speed_ms,0,blend_radius_m)
    |   movel([0.392601, -1.410802, -2.547453, -0.754134, 1.570796, 1.963398],accel_mss,speed_ms,0,blend_radius_m)
    |   movel([0.392818, -1.411188, -2.547164, -0.754038, 1.570796, 1.963614],accel_mss,speed_ms,0,blend_radius_m)
    |   movel([0.393019, -1.411582, -2.546868, -0.753940, 1.570796, 1.963815],accel_mss,speed_ms,0,blend_radius_m)
    |   movel([0.393205, -1.411984, -2.546565, -0.753840, 1.570796, 1.964002],accel_mss,speed_ms,0,blend_radius_m)
    |   movel([0.393378, -1.412398, -2.546254, -0.753738, 1.570796, 1.964174],accel_mss,speed_ms,0,blend_radius_m)
    |   movel([0.393536, -1.412818, -2.545937, -0.753634, 1.570796, 1.964332],accel_mss,speed_ms,0,blend_radius_m)
    |   movel([0.393679, -1.413248, -2.545613, -0.753528, 1.570796, 1.964475],accel_mss,speed_ms,0,blend_radius_m)
    |   movel([0.393805, -1.413685, -2.545283, -0.753421, 1.570796, 1.964601],accel_mss,speed_ms,0,blend_radius_m)
    |   movel([0.393919, -1.414134, -2.544944, -0.753311, 1.570796, 1.964715],accel_mss,speed_ms,0,blend_radius_m)
    |   movel([0.394015, -1.414592, -2.544598, -0.753199, 1.570796, 1.964811],accel_mss,speed_ms,0,blend_radius_m)
    |   movel([0.394098, -1.415057, -2.544247, -0.753086, 1.570796, 1.964894],accel_mss,speed_ms,0,blend_radius_m)
    |   movel([0.394161, -1.415529, -2.543889, -0.752971, 1.570796, 1.964957],accel_mss,speed_ms,0,blend_radius_m)
    |   movel([0.394208, -1.416008, -2.543526, -0.752855, 1.570796, 1.965005],accel_mss,speed_ms,0,blend_radius_m)
    |   movel([0.394244, -1.416527, -2.543132, -0.752730, 1.570796, 1.965041],accel_mss,speed_ms,0,blend_radius_m)
    |   movel([0.394266, -1.417051, -2.542735, -0.752604, 1.570796, 1.965062],accel_mss,speed_ms,0,blend_radius_m)
    |   movel([0.394270, -1.417580, -2.542332, -0.752477, 1.570796, 1.965067],accel_mss,speed_ms,0,blend_radius_m)
    |   movel([0.394263, -1.418111, -2.541928, -0.752350, 1.570796, 1.965060],accel_mss,speed_ms,0,blend_radius_m)
    |   movel([0.394240, -1.418648, -2.541519, -0.752222, 1.570796, 1.965037],accel_mss,speed_ms,0,blend_radius_m)
    |   movel([0.394198, -1.419317, -2.541008, -0.752063, 1.570796, 1.964994],accel_mss,speed_ms,0,blend_radius_m)
    |   movel([0.394143, -1.419990, -2.540495, -0.751904, 1.570796, 1.964939],accel_mss,speed_ms,0,blend_radius_m)
    |   movel([0.394072, -1.420667, -2.539977, -0.751745, 1.570796, 1.964869],accel_mss,speed_ms,0,blend_radius_m)
    |   movel([0.393990, -1.421345, -2.539458, -0.751586, 1.570796, 1.964787],accel_mss,speed_ms,0,blend_radius_m)
    |   movel([0.393894, -1.422025, -2.538937, -0.751427, 1.570796, 1.964690],accel_mss,speed_ms,0,blend_radius_m)
    |   movel([0.393714, -1.423197, -2.538037, -0.751156, 1.570796, 1.964510],accel_mss,speed_ms,0,blend_radius_m)
    |   movel([0.393522, -1.424369, -2.537134, -0.750886, 1.570796, 1.964318],accel_mss,speed_ms,0,blend_radius_m)
    |   movel([0.393320, -1.425543, -2.536228, -0.750618, 1.570796, 1.964116],accel_mss,speed_ms,0,blend_radius_m)
    |   movel([0.393108, -1.426716, -2.535322, -0.750352, 1.570796, 1.963904],accel_mss,speed_ms,0,blend_radius_m)
    |   movel([0.392787, -1.428496, -2.533941, -0.749952, 1.570796, 1.963583],accel_mss,speed_ms,0,blend_radius_m)
    |   movel([0.392487, -1.430267, -2.532563, -0.749559, 1.570796, 1.963283],accel_mss,speed_ms,0,blend_radius_m)
    |   movel([0.392236, -1.431866, -2.531314, -0.749209, 1.570796, 1.963033],accel_mss,speed_ms,0,blend_radius_m)
    |   movel([0.392009, -1.433455, -2.530070, -0.748864, 1.570796, 1.962805],accel_mss,speed_ms,0,blend_radius_m)
    |   movel([0.391837, -1.434816, -2.529000, -0.748572, 1.570796, 1.962634],accel_mss,speed_ms,0,blend_radius_m)
    |   movel([0.391687, -1.436167, -2.527937, -0.748285, 1.570796, 1.962483],accel_mss,speed_ms,0,blend_radius_m)
    |   movel([0.391601, -1.437205, -2.527117, -0.748066, 1.570796, 1.962397],accel_mss,speed_ms,0,blend_radius_m)
    |   movel([0.391551, -1.438230, -2.526307, -0.747852, 1.570796, 1.962347],accel_mss,speed_ms,0,blend_radius_m)
    |   movel([0.391508, -1.439583, -2.525235, -0.747572, 1.570796, 1.962305],accel_mss,speed_ms,0,blend_radius_m)
    |   movel([0.392550, -1.439260, -2.525491, -0.747638, 1.570796, 1.963346],accel_mss,speed_ms,0,blend_radius_m)
    |   movel([0.392795, -1.439189, -2.525547, -0.747653, 1.570796, 1.963591],accel_mss,speed_ms,0,blend_radius_m)
    |   movel([0.393037, -1.439128, -2.525596, -0.747666, 1.570796, 1.963834],accel_mss,speed_ms,0,blend_radius_m)
    |   movel([0.393281, -1.439079, -2.525634, -0.747676, 1.570796, 1.964078],accel_mss,speed_ms,0,blend_radius_m)
    |   movel([0.393521, -1.439039, -2.525666, -0.747684, 1.570796, 1.964318],accel_mss,speed_ms,0,blend_radius_m)
    |   movel([0.393758, -1.439012, -2.525688, -0.747690, 1.570796, 1.964555],accel_mss,speed_ms,0,blend_radius_m)
    |   movel([0.394097, -1.438985, -2.525709, -0.747695, 1.570796, 1.964893],accel_mss,speed_ms,0,blend_radius_m)
    |   movel([0.394430, -1.438971, -2.525720, -0.747698, 1.570796, 1.965226],accel_mss,speed_ms,0,blend_radius_m)
    |   movel([0.394757, -1.438971, -2.525720, -0.747698, 1.570796, 1.965553],accel_mss,speed_ms,0,blend_radius_m)
    |   movel([0.395081, -1.438982, -2.525711, -0.747696, 1.570796, 1.965877],accel_mss,speed_ms,0,blend_radius_m)
    |   movel([0.395399, -1.439008, -2.525691, -0.747690, 1.570796, 1.966195],accel_mss,speed_ms,0,blend_radius_m)
    |   movel([0.395710, -1.439046, -2.525661, -0.747682, 1.570796, 1.966506],accel_mss,speed_ms,0,blend_radius_m)
    |   movel([0.396014, -1.439097, -2.525620, -0.747672, 1.570796, 1.966811],accel_mss,speed_ms,0,blend_radius_m)
    |   movel([0.396309, -1.439162, -2.525569, -0.747658, 1.570796, 1.967105],accel_mss,speed_ms,0,blend_radius_m)
    |   movel([0.396510, -1.439216, -2.525526, -0.747647, 1.570796, 1.967307],accel_mss,speed_ms,0,blend_radius_m)
    |   movel([0.396703, -1.439280, -2.525475, -0.747634, 1.570796, 1.967499],accel_mss,speed_ms,0,blend_radius_m)
    |   movel([0.396887, -1.439355, -2.525416, -0.747619, 1.570796, 1.967683],accel_mss,speed_ms,0,blend_radius_m)
    |   movel([0.397064, -1.439440, -2.525348, -0.747601, 1.570796, 1.967860],accel_mss,speed_ms,0,blend_radius_m)
    |   movel([0.397232, -1.439535, -2.525272, -0.747581, 1.570796, 1.968029],accel_mss,speed_ms,0,blend_radius_m)
    |   movel([0.397450, -1.439677, -2.525160, -0.747552, 1.570796, 1.968246],accel_mss,speed_ms,0,blend_radius_m)
    |   movel([0.397652, -1.439833, -2.525036, -0.747520, 1.570796, 1.968448],accel_mss,speed_ms,0,blend_radius_m)
    |   movel([0.397839, -1.440004, -2.524900, -0.747485, 1.570796, 1.968635],accel_mss,speed_ms,0,blend_radius_m)
    |   movel([0.398012, -1.440187, -2.524755, -0.747447, 1.570796, 1.968808],accel_mss,speed_ms,0,blend_radius_m)
    |   movel([0.398169, -1.440382, -2.524600, -0.747407, 1.570796, 1.968965],accel_mss,speed_ms,0,blend_radius_m)
    |   movel([0.398323, -1.440605, -2.524423, -0.747361, 1.570796, 1.969119],accel_mss,speed_ms,0,blend_radius_m)
    |   movel([0.398461, -1.440837, -2.524238, -0.747314, 1.570796, 1.969257],accel_mss,speed_ms,0,blend_radius_m)
    |   movel([0.398587, -1.441078, -2.524046, -0.747265, 1.570796, 1.969383],accel_mss,speed_ms,0,blend_radius_m)
    |   movel([0.398695, -1.441329, -2.523847, -0.747214, 1.570796, 1.969491],accel_mss,speed_ms,0,blend_radius_m)
    |   movel([0.398791, -1.441588, -2.523640, -0.747161, 1.570796, 1.969587],accel_mss,speed_ms,0,blend_radius_m)
    |   movel([0.398873, -1.441855, -2.523428, -0.747107, 1.570796, 1.969669],accel_mss,speed_ms,0,blend_radius_m)
    |   movel([0.398938, -1.442130, -2.523209, -0.747051, 1.570796, 1.969734],accel_mss,speed_ms,0,blend_radius_m)
    |   movel([0.398988, -1.442410, -2.522984, -0.746994, 1.570796, 1.969784],accel_mss,speed_ms,0,blend_radius_m)
    |   movel([0.399023, -1.442699, -2.522754, -0.746936, 1.570796, 1.969819],accel_mss,speed_ms,0,blend_radius_m)
    |   movel([0.399043, -1.442992, -2.522520, -0.746877, 1.570796, 1.969839],accel_mss,speed_ms,0,blend_radius_m)
    |   movel([0.399045, -1.443272, -2.522296, -0.746821, 1.570796, 1.969842],accel_mss,speed_ms,0,blend_radius_m)
    |   movel([0.399031, -1.443556, -2.522069, -0.746764, 1.570796, 1.969827],accel_mss,speed_ms,0,blend_radius_m)
    |   movel([0.398997, -1.443846, -2.521838, -0.746706, 1.570796, 1.969793],accel_mss,speed_ms,0,blend_radius_m)
    |   movel([0.398949, -1.444137, -2.521605, -0.746648, 1.570796, 1.969745],accel_mss,speed_ms,0,blend_radius_m)
    |   movel([0.398881, -1.444434, -2.521367, -0.746588, 1.570796, 1.969677],accel_mss,speed_ms,0,blend_radius_m)
    |   movel([0.398791, -1.444752, -2.521112, -0.746525, 1.570796, 1.969587],accel_mss,speed_ms,0,blend_radius_m)
    |   movel([0.398685, -1.445073, -2.520855, -0.746462, 1.570796, 1.969481],accel_mss,speed_ms,0,blend_radius_m)
    |   movel([0.398564, -1.445394, -2.520597, -0.746398, 1.570796, 1.969360],accel_mss,speed_ms,0,blend_radius_m)
    |   movel([0.398430, -1.445714, -2.520340, -0.746335, 1.570796, 1.969226],accel_mss,speed_ms,0,blend_radius_m)
    |   movel([0.398279, -1.446034, -2.520083, -0.746272, 1.570796, 1.969075],accel_mss,speed_ms,0,blend_radius_m)
    |   movel([0.398113, -1.446354, -2.519826, -0.746209, 1.570796, 1.968909],accel_mss,speed_ms,0,blend_radius_m)
    |   movel([0.397933, -1.446671, -2.519571, -0.746147, 1.570796, 1.968729],accel_mss,speed_ms,0,blend_radius_m)
    |   movel([0.397740, -1.446984, -2.519319, -0.746086, 1.570796, 1.968537],accel_mss,speed_ms,0,blend_radius_m)
    |   movel([0.397534, -1.447294, -2.519069, -0.746025, 1.570796, 1.968330],accel_mss,speed_ms,0,blend_radius_m)
    |   movel([0.397314, -1.447600, -2.518823, -0.745966, 1.570796, 1.968110],accel_mss,speed_ms,0,blend_radius_m)
    |   movel([0.397082, -1.447900, -2.518581, -0.745908, 1.570796, 1.967879],accel_mss,speed_ms,0,blend_radius_m)
    |   movel([0.396837, -1.448197, -2.518342, -0.745850, 1.570796, 1.967633],accel_mss,speed_ms,0,blend_radius_m)
    |   movel([0.396579, -1.448488, -2.518107, -0.745794, 1.570796, 1.967375],accel_mss,speed_ms,0,blend_radius_m)
    |   movel([0.396311, -1.448772, -2.517877, -0.745740, 1.570796, 1.967108],accel_mss,speed_ms,0,blend_radius_m)
    |   movel([0.396035, -1.449048, -2.517655, -0.745687, 1.570796, 1.966831],accel_mss,speed_ms,0,blend_radius_m)
    |   movel([0.395748, -1.449317, -2.517437, -0.745635, 1.570796, 1.966544],accel_mss,speed_ms,0,blend_radius_m)
    |   movel([0.395451, -1.449576, -2.517227, -0.745585, 1.570796, 1.966247],accel_mss,speed_ms,0,blend_radius_m)
    |   movel([0.395144, -1.449829, -2.517023, -0.745537, 1.570796, 1.965940],accel_mss,speed_ms,0,blend_radius_m)
    |   movel([0.394831, -1.450071, -2.516827, -0.745491, 1.570796, 1.965627],accel_mss,speed_ms,0,blend_radius_m)
    |   movel([0.394509, -1.450305, -2.516637, -0.745446, 1.570796, 1.965305],accel_mss,speed_ms,0,blend_radius_m)
    |   movel([0.394181, -1.450529, -2.516456, -0.745404, 1.570796, 1.964977],accel_mss,speed_ms,0,blend_radius_m)
    |   movel([0.393847, -1.450742, -2.516283, -0.745364, 1.570796, 1.964643],accel_mss,speed_ms,0,blend_radius_m)
    |   movel([0.393506, -1.450945, -2.516119, -0.745325, 1.570796, 1.964303],accel_mss,speed_ms,0,blend_radius_m)
    |   movel([0.393161, -1.451135, -2.515964, -0.745289, 1.570796, 1.963957],accel_mss,speed_ms,0,blend_radius_m)
    |   movel([0.392812, -1.451314, -2.515820, -0.745256, 1.570796, 1.963608],accel_mss,speed_ms,0,blend_radius_m)
    |   movel([0.392460, -1.451480, -2.515685, -0.745224, 1.570796, 1.963257],accel_mss,speed_ms,0,blend_radius_m)
    |   movel([0.392104, -1.451635, -2.515559, -0.745195, 1.570796, 1.962901],accel_mss,speed_ms,0,blend_radius_m)
    |   movel([0.391748, -1.451777, -2.515444, -0.745168, 1.570796, 1.962545],accel_mss,speed_ms,0,blend_radius_m)
    |   movel([0.391417, -1.451896, -2.515347, -0.745146, 1.570796, 1.962213],accel_mss,speed_ms,0,blend_radius_m)
    |   movel([0.391083, -1.452003, -2.515260, -0.745126, 1.570796, 1.961879],accel_mss,speed_ms,0,blend_radius_m)
    |   movel([0.390903, -1.452053, -2.515220, -0.745117, 1.570796, 1.961700],accel_mss,speed_ms,0,blend_radius_m)
    |   movel([0.390725, -1.452094, -2.515186, -0.745109, 1.570796, 1.961522],accel_mss,speed_ms,0,blend_radius_m)
    |   movel([0.390547, -1.452127, -2.515159, -0.745103, 1.570796, 1.961343],accel_mss,speed_ms,0,blend_radius_m)
    |   movel([0.390347, -1.452154, -2.515138, -0.745098, 1.570796, 1.961144],accel_mss,speed_ms,0,blend_radius_m)
    |   movel([0.390151, -1.452172, -2.515122, -0.745094, 1.570796, 1.960948],accel_mss,speed_ms,0,blend_radius_m)
    |   movel([0.389957, -1.452183, -2.515114, -0.745092, 1.570796, 1.960753],accel_mss,speed_ms,0,blend_radius_m)
    |   movel([0.389519, -1.452193, -2.515105, -0.745090, 1.570796, 1.960315],accel_mss,speed_ms,0,blend_radius_m)
    |   movel([0.389085, -1.452194, -2.515105, -0.745090, 1.570796, 1.959881],accel_mss,speed_ms,0,blend_radius_m)
    |   movel([0.388657, -1.452187, -2.515111, -0.745092, 1.570796, 1.959453],accel_mss,speed_ms,0,blend_radius_m)
    |   movel([0.388232, -1.452172, -2.515123, -0.745094, 1.570796, 1.959028],accel_mss,speed_ms,0,blend_radius_m)
    |   movel([0.388045, -1.452160, -2.515132, -0.745097, 1.570796, 1.958841],accel_mss,speed_ms,0,blend_radius_m)
    |   movel([0.387864, -1.452138, -2.515150, -0.745101, 1.570796, 1.958660],accel_mss,speed_ms,0,blend_radius_m)
    |   movel([0.387687, -1.452109, -2.515174, -0.745106, 1.570796, 1.958483],accel_mss,speed_ms,0,blend_radius_m)
    |   movel([0.387532, -1.452075, -2.515201, -0.745113, 1.570796, 1.958328],accel_mss,speed_ms,0,blend_radius_m)
    |   movel([0.387386, -1.452031, -2.515237, -0.745121, 1.570796, 1.958183],accel_mss,speed_ms,0,blend_radius_m)
    |   movel([0.387246, -1.451980, -2.515279, -0.745130, 1.570796, 1.958043],accel_mss,speed_ms,0,blend_radius_m)
    |   movel([0.386998, -1.451870, -2.515368, -0.745151, 1.570796, 1.957795],accel_mss,speed_ms,0,blend_radius_m)
    |   movel([0.386762, -1.451749, -2.515467, -0.745174, 1.570796, 1.957558],accel_mss,speed_ms,0,blend_radius_m)
    |   movel([0.386519, -1.451600, -2.515587, -0.745202, 1.570796, 1.957316],accel_mss,speed_ms,0,blend_radius_m)
    |   movel([0.386289, -1.451440, -2.515717, -0.745232, 1.570796, 1.957085],accel_mss,speed_ms,0,blend_radius_m)
    |   movel([0.386074, -1.451266, -2.515859, -0.745265, 1.570796, 1.956871],accel_mss,speed_ms,0,blend_radius_m)
    |   movel([0.385874, -1.451079, -2.516010, -0.745300, 1.570796, 1.956670],accel_mss,speed_ms,0,blend_radius_m)
    |   movel([0.385688, -1.450878, -2.516173, -0.745338, 1.570796, 1.956484],accel_mss,speed_ms,0,blend_radius_m)
    |   movel([0.385519, -1.450666, -2.516345, -0.745378, 1.570796, 1.956316],accel_mss,speed_ms,0,blend_radius_m)
    |   movel([0.385367, -1.450440, -2.516528, -0.745421, 1.570796, 1.956163],accel_mss,speed_ms,0,blend_radius_m)
    |   movel([0.385232, -1.450203, -2.516720, -0.745466, 1.570796, 1.956029],accel_mss,speed_ms,0,blend_radius_m)
    |   movel([0.385113, -1.449955, -2.516921, -0.745513, 1.570796, 1.955909],accel_mss,speed_ms,0,blend_radius_m)
    |   movel([0.385013, -1.449698, -2.517129, -0.745562, 1.570796, 1.955809],accel_mss,speed_ms,0,blend_radius_m)
    |   movel([0.384927, -1.449430, -2.517346, -0.745613, 1.570796, 1.955724],accel_mss,speed_ms,0,blend_radius_m)
    |   movel([0.384859, -1.449151, -2.517571, -0.745667, 1.570796, 1.955655],accel_mss,speed_ms,0,blend_radius_m)
    |   movel([0.384811, -1.448865, -2.517802, -0.745722, 1.570796, 1.955608],accel_mss,speed_ms,0,blend_radius_m)
    |   movel([0.384780, -1.448570, -2.518040, -0.745778, 1.570796, 1.955576],accel_mss,speed_ms,0,blend_radius_m)
    |   movel([0.384766, -1.448269, -2.518283, -0.745836, 1.570796, 1.955562],accel_mss,speed_ms,0,blend_radius_m)
    |   movel([0.384772, -1.447962, -2.518531, -0.745896, 1.570796, 1.955568],accel_mss,speed_ms,0,blend_radius_m)
    |   movel([0.384793, -1.447649, -2.518784, -0.745957, 1.570796, 1.955589],accel_mss,speed_ms,0,blend_radius_m)
    |   movel([0.384836, -1.447331, -2.519039, -0.746018, 1.570796, 1.955632],accel_mss,speed_ms,0,blend_radius_m)
    |   movel([0.384893, -1.447009, -2.519299, -0.746081, 1.570796, 1.955689],accel_mss,speed_ms,0,blend_radius_m)
    |   movel([0.384971, -1.446683, -2.519561, -0.746145, 1.570796, 1.955767],accel_mss,speed_ms,0,blend_radius_m)
    |   movel([0.385066, -1.446353, -2.519827, -0.746209, 1.570796, 1.955862],accel_mss,speed_ms,0,blend_radius_m)
    |   movel([0.385177, -1.446021, -2.520094, -0.746275, 1.570796, 1.955973],accel_mss,speed_ms,0,blend_radius_m)
    |   movel([0.385307, -1.445688, -2.520361, -0.746340, 1.570796, 1.956103],accel_mss,speed_ms,0,blend_radius_m)
    |   movel([0.385453, -1.445353, -2.520630, -0.746406, 1.570796, 1.956250],accel_mss,speed_ms,0,blend_radius_m)
    |   movel([0.385616, -1.445020, -2.520897, -0.746472, 1.570796, 1.956413],accel_mss,speed_ms,0,blend_radius_m)
    |   movel([0.385796, -1.444689, -2.521162, -0.746538, 1.570796, 1.956592],accel_mss,speed_ms,0,blend_radius_m)
    |   movel([0.385990, -1.444358, -2.521427, -0.746603, 1.570796, 1.956786],accel_mss,speed_ms,0,blend_radius_m)
    |   movel([0.386200, -1.444031, -2.521689, -0.746669, 1.570796, 1.956996],accel_mss,speed_ms,0,blend_radius_m)
    |   movel([0.386426, -1.443708, -2.521948, -0.746733, 1.570796, 1.957222],accel_mss,speed_ms,0,blend_radius_m)
    |   movel([0.386666, -1.443387, -2.522205, -0.746798, 1.570796, 1.957462],accel_mss,speed_ms,0,blend_radius_m)
    |   movel([0.386921, -1.443072, -2.522457, -0.746861, 1.570796, 1.957717],accel_mss,speed_ms,0,blend_radius_m)
    |   movel([0.387188, -1.442763, -2.522703, -0.746923, 1.570796, 1.957984],accel_mss,speed_ms,0,blend_radius_m)
    |   movel([0.387468, -1.442460, -2.522945, -0.746984, 1.570796, 1.958264],accel_mss,speed_ms,0,blend_radius_m)
    |   movel([0.387758, -1.442165, -2.523180, -0.747044, 1.570796, 1.958554],accel_mss,speed_ms,0,blend_radius_m)
    |   movel([0.388062, -1.441876, -2.523411, -0.747102, 1.570796, 1.958859],accel_mss,speed_ms,0,blend_radius_m)
    |   movel([0.388376, -1.441596, -2.523634, -0.747159, 1.570796, 1.959173],accel_mss,speed_ms,0,blend_radius_m)
    |   movel([0.388701, -1.441326, -2.523849, -0.747214, 1.570796, 1.959497],accel_mss,speed_ms,0,blend_radius_m)
